// TwinCAT 3 PLC project Motion
// ProgramVersion: 3.1.4022.7
// libraries:
//   LCLS General, * (SLAC)
//   lcls-twincat-motion, * (SLAC)
//   PMPS, * (SLAC - LCLS)
//   Tc2_MC2, * (Beckhoff Automation GmbH)
//   Tc2_Standard, * (Beckhoff Automation GmbH)
//   Tc2_System, * (Beckhoff Automation GmbH)
//   Tc3_Module, * (Beckhoff Automation GmbH)
//   TcUnit, * (www.tcunit.org)
// project tree:
//   DUTs/ DUT_SensorHGS.TcDUT, DUT_Sensor.TcDUT (not stored)
//   GVLs/ GVL_Main.TcGVL, GVL_PMPS.TcGVL, GVL_Sensor.TcGVL (not stored)
//   / PlcTask.TcTTO
//   POUs/ FB_2AxesTrans.TcPOU, FB_3AxesJack.TcPOU, PRG1_MAIN_PlcTask.TcPOU, FB_Slits.TcPOU, PRG_2Theta.TcPOU, PRG_DET_ARM.TcPOU, PRG_DET_CHAMBER.TcPOU, PRG_DET_SLIT.TcPOU, PRG_DET_FRAME.TcPOU, PRG_OPT.TcPOU, PRG_OPT_XPM.TcPOU, PRG_OPT_SLITS.TcPOU, PRG_OPT_YG.TcPOU, PRG_Sensor.TcPOU
// real-time tasks:
//   TASK PlcTask: cycle T#10ms, priority 20, ADS port 350
// motion (NC):
//   TASK NC-Task 1 SAF: cycle T#2ms, priority 4, ADS port 501
//   TASK NC-Task 1 SVB: cycle T#10ms, priority 8, ADS port 511
//   AXIS ServoDrive (id 1)
//     General: UnitName=deg
//     Dynamic: AccelerationMaximum=10, DecelerationMaximum=10, Acceleration=0.5, Deceleration=0.5, Jerk=1
//     Velo: RefSearch=0.25, RefSync=0.25, SlowManual=0.25, FastManual=0.25, Maximum=0.25
//     OtherSettings: AllowMotionCmdToSlave=true, PulseDistancePos=1, PulseDistanceNeg=1
//     encoder EncType=19
//       EncPara: ScaleFactorNumerator=3.001664895e-06, Offset=-76.2211171, MaxCount=#xffffffff
//         SoftEndMinControl: Enable=true, Range=42
//         SoftEndMaxControl: Enable=true, Range=149.4
//     drive DrvType=16
//       DrvPara: MaxCount=#xffffffff, DriveControlDWord=#x00020100
//         Analog: VeloReferenz=0.25, ScaleFactorActTorque=0.1
//         TimeComp: TaskDelayCycles=1
//     controller CtrType=2
//       CtrPara: PriorControlFactor=1
//         PosDiffControl: Range=2
//         PID: DeadBandPosition=0.05
//         Observer: BandWidth=20
//   AXIS Stepper (id 27)
//     General: UnitName=deg
//     Dynamic: AccelerationMaximum=1.5, DecelerationMaximum=1.5, Acceleration=1.4, Deceleration=0.7, Jerk=2.8
//     Velo: Maximum=0.7
//     PositionAreaControl: Range=0.5
//     TargetPosControl: Range=0.1
//     OtherSettings: AllowMotionCmdToSlave=true
//     encoder EncType=29
//       EncPara: ScaleFactorNumerator=3.001664895e-06, Offset=13.6052237, MaxCount=#xffffffff
//         SoftEndMinControl: Enable=true, Range=42
//         SoftEndMaxControl: Enable=true, Range=149.4
//         Inc: RefSoftSyncMask=#x0000ffff
//     drive DrvType=24
//       Analog: VeloReferenz=0.715862885, ScaleFactorActTorque=0.1
//       TimeComp: TaskDelayCycles=1
//     controller CtrType=2
//       CtrPara: PriorControlFactor=1
//         PosDiffControl: Range=0.5
//         PID: DeadBandPosition=0.05
//         Observer: BandWidth=20
//   AXIS XS1 (id 11)
//     Dynamic: AccelerationMaximum=20, DecelerationMaximum=20, Acceleration=10, Deceleration=10, Jerk=100
//     Velo: Maximum=1
//     PositionAreaControl: Range=1
//     TargetPosControl: Range=0.05
//     OtherSettings: AllowMotionCmdToSlave=true
//     encoder EncType=29
//       EncPara: ScaleFactorNumerator=5e-05, Offset=-48.701, MaxCount=#xffffffff
//         SoftEndMinControl: Enable=true, Range=-25
//         SoftEndMaxControl: Enable=true, Range=25
//         Inc: RefSoftSyncMask=#x0000ffff
//     drive DrvType=24
//       Analog: VeloReferenz=1, ScaleFactorActTorque=0.1
//       TimeComp: TaskDelayCycles=1
//     controller CtrType=2
//       CtrPara: PriorControlFactor=1
//         PosDiffControl: Range=1
//         PID: DeadBandPosition=0.0002
//         Observer: BandWidth=20
//   AXIS XS2 (id 12)
//     Dynamic: AccelerationMaximum=20, DecelerationMaximum=20, Acceleration=10, Deceleration=10, Jerk=100
//     Velo: Maximum=1
//     PositionAreaControl: Range=1
//     TargetPosControl: Range=0.05
//     OtherSettings: AllowMotionCmdToSlave=true
//     encoder EncType=29
//       EncPara: ScaleFactorNumerator=5e-05, Offset=-50.138, MaxCount=#xffffffff
//         SoftEndMinControl: Enable=true, Range=-25
//         SoftEndMaxControl: Enable=true, Range=25
//         Inc: RefSoftSyncMask=#x0000ffff
//     drive DrvType=24
//       Analog: VeloReferenz=1, ScaleFactorActTorque=0.1
//       TimeComp: TaskDelayCycles=1
//     controller CtrType=2
//       CtrPara: PriorControlFactor=1
//         PosDiffControl: Range=1
//         PID: DeadBandPosition=0.0002
//         Observer: BandWidth=20
//   AXIS YS1 (id 13)
//     Dynamic: AccelerationMaximum=20, DecelerationMaximum=20, Acceleration=10, Deceleration=10, Jerk=100
//     Velo: Maximum=1
//     PositionAreaControl: Range=1
//     TargetPosControl: Range=0.05
//     OtherSettings: AllowMotionCmdToSlave=true
//     encoder EncType=29
//       EncPara: ScaleFactorNumerator=5e-05, Offset=-53.276, MaxCount=#xffffffff
//         SoftEndMinControl: Enable=true, Range=-25
//         SoftEndMaxControl: Enable=true, Range=25
//         Inc: RefSoftSyncMask=#x0000ffff
//     drive DrvType=24
//       Analog: VeloReferenz=1, ScaleFactorActTorque=0.1
//       TimeComp: TaskDelayCycles=1
//     controller CtrType=2
//       CtrPara: PriorControlFactor=1
//         PosDiffControl: Range=1
//         PID: DeadBandPosition=0.0002
//         Observer: BandWidth=20
//   AXIS YS2 (id 14)
//     Dynamic: AccelerationMaximum=20, DecelerationMaximum=20, Acceleration=10, Deceleration=10, Jerk=100
//     Velo: Maximum=1
//     PositionAreaControl: Range=1
//     TargetPosControl: Range=0.05
//     OtherSettings: AllowMotionCmdToSlave=true
//     encoder EncType=29
//       EncPara: ScaleFactorNumerator=5e-05, Offset=-50.673, MaxCount=#xffffffff
//         SoftEndMinControl: Enable=true, Range=-25
//         SoftEndMaxControl: Enable=true, Range=25
//         Inc: RefSoftSyncMask=#x0000ffff
//     drive DrvType=24
//       Analog: VeloReferenz=1, ScaleFactorActTorque=0.1
//       TimeComp: TaskDelayCycles=1
//     controller CtrType=2
//       CtrPara: PriorControlFactor=1
//         PosDiffControl: Range=1
//         PID: DeadBandPosition=0.0002
//         Observer: BandWidth=20
//   AXIS YG1 (id 17)
//     Dynamic: AccelerationMaximum=0.4, DecelerationMaximum=0.4, Acceleration=0.2, Deceleration=0.2, Jerk=0.4
//     Velo: SlowManual=0.25, FastManual=0.5, Maximum=0.05
//     PositionAreaControl: Range=0.1
//     TargetPosControl: Range=0.05
//     BacklashCompensation: Range=0.025
//     OtherSettings: AllowMotionCmdToSlave=true, PulseDistancePos=1, PulseDistanceNeg=1
//     encoder EncType=29
//       EncPara: ScaleFactorNumerator=5e-06, Offset=-48.289375, MaxCount=#xffffffff
//         SoftEndMinControl: Enable=true, Range=-7.2
//         SoftEndMaxControl: Enable=true, Range=7.2
//         Inc: RefSoftSyncMask=#x0000ffff
//     drive DrvType=24
//       Analog: VeloReferenz=0.1, ScaleFactorActTorque=0.1
//       TimeComp: TaskDelayCycles=1
//     controller CtrType=2
//       CtrPara: PriorControlFactor=1
//         PosDiffControl: Range=2
//         PID: DeadBandPosition=0.0001
//         Observer: BandWidth=20
//   AXIS YG2 (id 18)
//     Dynamic: AccelerationMaximum=0.4, DecelerationMaximum=0.4, Acceleration=0.2, Deceleration=0.2, Jerk=0.4
//     Velo: Maximum=0.05
//     PositionAreaControl: Range=0.5
//     TargetPosControl: Range=0.05
//     OtherSettings: AllowMotionCmdToSlave=true
//     encoder EncType=29
//       EncPara: ScaleFactorNumerator=5e-06, Offset=-49.0846, MaxCount=#xffffffff
//         SoftEndMinControl: Enable=true, Range=-7.2
//         SoftEndMaxControl: Enable=true, Range=-7.2
//         Inc: RefSoftSyncMask=#x0000ffff
//     drive DrvType=24
//       Analog: VeloReferenz=0.1, ScaleFactorActTorque=0.1
//       TimeComp: TaskDelayCycles=1
//     controller CtrType=2
//       CtrPara: PriorControlFactor=1
//         PosDiffControl: Range=2
//         PID: DeadBandPosition=0.0001
//         Observer: BandWidth=20
//   AXIS YG3 (id 19)
//     Dynamic: AccelerationMaximum=0.4, DecelerationMaximum=0.4, Acceleration=0.2, Deceleration=0.2, Jerk=0.4
//     Velo: Maximum=0.05
//     PositionAreaControl: Range=0.1
//     TargetPosControl: Range=0.05
//     OtherSettings: AllowMotionCmdToSlave=true
//     encoder EncType=29
//       EncPara: ScaleFactorNumerator=5e-06, Offset=-49.5733, MaxCount=#xffffffff
//         SoftEndMinControl: Enable=true, Range=-7.2
//         SoftEndMaxControl: Enable=true, Range=7.2
//         Inc: RefSoftSyncMask=#x0000ffff
//     drive DrvType=24
//       Analog: VeloReferenz=0.1, ScaleFactorActTorque=0.1
//       TimeComp: TaskDelayCycles=1
//     controller CtrType=2
//       CtrPara: PriorControlFactor=1
//         PosDiffControl: Range=2
//         PID: DeadBandPosition=0.0001
//         Observer: BandWidth=20
//   AXIS RxG (id 15)
//     General: UnitName=mrad
//     Dynamic: AccelerationMaximum=2, DecelerationMaximum=2, Acceleration=2, Deceleration=2, Jerk=10
//     Velo: Maximum=1.29
//     TargetPosControl: Range=0.01
//     OtherSettings: AllowMotionCmdToSlave=true
//     encoder EncType=19
//       EncPara: ScaleFactorNumerator=1.462918079, ScaleFactorDenominator=1000000, Offset=2351.695, MaxCount=#xffffffff
//         SoftEndMinControl: Enable=true, Range=-17.5
//         SoftEndMaxControl: Enable=true, Range=87.5
//         Inc: RefSoftSyncMask=#x0000ffff
//     drive DrvType=24
//       Analog: VeloReferenz=1.29032258064516, ScaleFactorActTorque=0.1
//       TimeComp: TaskDelayCycles=1
//     controller CtrType=2
//       CtrPara: PriorControlFactor=1
//         PosDiffControl: Range=0.5
//         PID: DeadBandPosition=5e-05
//         Observer: BandWidth=20
//   AXIS XG (id 16)
//     Dynamic: AccelerationMaximum=40, DecelerationMaximum=40, Acceleration=20, Deceleration=20, Jerk=20000
//     Velo: Maximum=2
//     TargetPosControl: Range=0.1
//     OtherSettings: AllowMotionCmdToSlave=true
//     encoder EncType=29
//       EncPara: ScaleFactorNumerator=5e-05, Offset=-123.91085, MaxCount=#xffffffff
//         SoftEndMinControl: Enable=true, Range=-95
//         SoftEndMaxControl: Enable=true, Range=95
//         Inc: RefSoftSyncMask=#x0000ffff
//     drive DrvType=24
//       Analog: VeloReferenz=10, ScaleFactorActTorque=0.1
//       TimeComp: TaskDelayCycles=1
//     controller CtrType=2
//       CtrPara: PriorControlFactor=1
//         PID: DeadBandPosition=0.001
//         Observer: BandWidth=20
//   AXIS XPM1 (id 20)
//     Dynamic: AccelerationMaximum=20, DecelerationMaximum=20, Acceleration=20, Deceleration=20, Jerk=400
//     Velo: RefSearch=1, RefSync=1, SlowManual=0.5, FastManual=1, Maximum=0.1
//     PositionAreaControl: Range=1
//     TargetPosControl: Range=0.02
//     OtherSettings: AllowMotionCmdToSlave=true, PulseDistancePos=1, PulseDistanceNeg=1
//     encoder EncType=29
//       EncPara: ScaleFactorNumerator=5e-05, Offset=-50.788, MaxCount=#xffffffff
//         SoftEndMinControl: Enable=true, Range=-17.5
//         SoftEndMaxControl: Enable=true, Range=17.5
//         Inc: RefSoftSyncMask=#x0000ffff
//     drive DrvType=24
//       Analog: VeloReferenz=0.2, ScaleFactorActTorque=0.1
//       TimeComp: TaskDelayCycles=1
//     controller CtrType=2
//       CtrPara: PriorControlFactor=1
//         PosDiffControl: Range=0.5, Time=0.01
//         PID: DeadBandPosition=0.0001
//         Observer: BandWidth=20
//   AXIS XPM2 (id 21)
//     Dynamic: AccelerationMaximum=20, DecelerationMaximum=20, Acceleration=20, Deceleration=20, Jerk=400
//     Velo: RefSearch=1, RefSync=1, SlowManual=0.5, FastManual=1, Maximum=0.1
//     PositionAreaControl: Range=1
//     TargetPosControl: Range=0.02
//     OtherSettings: AllowMotionCmdToSlave=true, PulseDistancePos=1, PulseDistanceNeg=1
//     encoder EncType=29
//       EncPara: ScaleFactorNumerator=5e-05, Offset=-48.577, MaxCount=#xffffffff
//         SoftEndMinControl: Enable=true, Range=-17.5
//         SoftEndMaxControl: Enable=true, Range=17.5
//         Inc: RefSoftSyncMask=#x0000ffff
//     drive DrvType=24
//       Analog: VeloReferenz=0.2, ScaleFactorActTorque=0.1
//       TimeComp: TaskDelayCycles=1
//     controller CtrType=2
//       CtrPara: PriorControlFactor=1
//         PosDiffControl: Range=1
//         PID: DeadBandPosition=0.0001
//         Observer: BandWidth=20
//   AXIS RzPM (id 22)
//     General: UnitName=mrad
//     Dynamic: AccelerationMaximum=2.6, DecelerationMaximum=2.6, Acceleration=2.6, Deceleration=2.6, Jerk=52
//     Velo: RefSearch=2000, RefSync=2000, SlowManual=1000, FastManual=2000, Maximum=0.2
//     PositionAreaControl: Range=0.1
//     TargetPosControl: Range=0.01
//     OtherSettings: AllowMotionCmdToSlave=true
//     encoder EncType=29
//       EncPara: ScaleFactorNumerator=0.299580587, ScaleFactorDenominator=1000, Offset=-205.8664, MaxCount=#xffffffff
//         SoftEndMinControl: Enable=true, Range=-60
//         SoftEndMaxControl: Enable=true, Range=60
//         Inc: RefSoftSyncMask=#x0000ffff
//     drive DrvType=24
//       Analog: VeloReferenz=1.3333333, ScaleFactorActTorque=0.1
//       TimeComp: TaskDelayCycles=1
//     controller CtrType=2
//       CtrPara: PriorControlFactor=1
//         PosDiffControl: Range=0.1
//         PID: DeadBandPosition=0.0005
//         Observer: BandWidth=20
//   AXIS YDF1 (id 23)
//     Dynamic: AccelerationMaximum=1, DecelerationMaximum=1, Acceleration=0.8, Deceleration=0.8, Jerk=3.2
//     Velo: FastManual=0, Maximum=0.05
//     PositionAreaControl: Range=0.5
//     OtherSettings: AllowMotionCmdToSlave=true
//     encoder EncType=1
//       EncPara: ScaleFactorNumerator=1
//         SoftEndMinControl: Enable=true, Range=-0.5
//         SoftEndMaxControl: Range=21.5
//         Inc: RefSoftSyncMask=#x0000ffff
//     drive DrvType=24
//       Analog: VeloReferenz=0.333336, ScaleFactorActTorque=0.1
//       TimeComp: TaskDelayCycles=1
//     controller CtrType=1
//       CtrPara: PriorControlFactor=1
//         PosDiffControl: Range=0.5
//         Observer: BandWidth=20
//   AXIS YDF2 (id 24)
//     Dynamic: AccelerationMaximum=1, DecelerationMaximum=1, Acceleration=0.8, Deceleration=0.8, Jerk=3.2
//     Velo: FastManual=0, Maximum=0.05
//     PositionAreaControl: Range=0.5
//     OtherSettings: AllowMotionCmdToSlave=true
//     encoder EncType=1
//       EncPara: ScaleFactorNumerator=4.2e-05
//         SoftEndMinControl: Enable=true, Range=-0.5
//         SoftEndMaxControl: Range=21.5
//         Inc: RefSoftSyncMask=#x0000ffff
//     drive DrvType=24
//       Analog: VeloReferenz=0.333336, ScaleFactorActTorque=0.1
//       TimeComp: TaskDelayCycles=1
//     controller CtrType=1
//       CtrPara: PriorControlFactor=1
//         PosDiffControl: Range=0.5
//         Observer: BandWidth=20
//   AXIS YDF3 (id 25)
//     Dynamic: AccelerationMaximum=1, DecelerationMaximum=1, Acceleration=0.8, Deceleration=0.8, Jerk=3.2
//     Velo: FastManual=0, Maximum=0.05
//     PositionAreaControl: Range=0.5
//     OtherSettings: AllowMotionCmdToSlave=true
//     encoder EncType=1
//       EncPara: ScaleFactorNumerator=4.2e-05
//         SoftEndMinControl: Enable=true, Range=-0.5
//         SoftEndMaxControl: Enable=true, Range=21.5
//         Inc: RefSoftSyncMask=#x0000ffff
//     drive DrvType=24
//       Analog: VeloReferenz=0.333336, ScaleFactorActTorque=0.1
//       TimeComp: TaskDelayCycles=1
//     controller CtrType=1
//       CtrPara: PriorControlFactor=1
//         PosDiffControl: Range=0.5
//         Observer: BandWidth=20
//   AXIS XSDC1 (id 2)
//     Dynamic: AccelerationMaximum=20, DecelerationMaximum=20, Acceleration=10, Deceleration=10, Jerk=100
//     Velo: Maximum=1
//     PositionAreaControl: Range=1
//     TargetPosControl: Range=0.1
//     OtherSettings: AllowMotionCmdToSlave=true
//     encoder EncType=29
//       EncPara: ScaleFactorNumerator=5e-05, Offset=-49.035, MaxCount=#xffffffff
//         SoftEndMinControl: Enable=true, Range=-25
//         SoftEndMaxControl: Enable=true, Range=25
//         Inc: RefSoftSyncMask=#x0000ffff
//     drive DrvType=24
//       Analog: VeloReferenz=1, ScaleFactorActTorque=0.1
//       TimeComp: TaskDelayCycles=1
//     controller CtrType=2
//       CtrPara: PriorControlFactor=1
//         PosDiffControl: Range=1
//         PID: DeadBandPosition=0.0002
//         Observer: BandWidth=20
//   AXIS XSDC2 (id 3)
//     Dynamic: AccelerationMaximum=20, DecelerationMaximum=20, Acceleration=10, Deceleration=10, Jerk=100
//     Velo: Maximum=1
//     PositionAreaControl: Range=1
//     TargetPosControl: Range=0.1
//     OtherSettings: AllowMotionCmdToSlave=true
//     encoder EncType=29
//       EncPara: ScaleFactorNumerator=5e-05, Offset=-49.27, MaxCount=#xffffffff
//         SoftEndMinControl: Enable=true, Range=-25
//         SoftEndMaxControl: Enable=true, Range=25
//         Inc: RefSoftSyncMask=#x0000ffff
//     drive DrvType=24
//       Analog: VeloReferenz=1, ScaleFactorActTorque=0.1
//       TimeComp: TaskDelayCycles=1
//     controller CtrType=2
//       CtrPara: PriorControlFactor=1
//         PosDiffControl: Range=1
//         PID: DeadBandPosition=0.0002
//         Observer: BandWidth=20
//   AXIS YSDC1 (id 4)
//     Dynamic: AccelerationMaximum=20, DecelerationMaximum=20, Acceleration=10, Deceleration=10, Jerk=100
//     Velo: Maximum=1
//     PositionAreaControl: Range=1
//     TargetPosControl: Range=0.1
//     OtherSettings: AllowMotionCmdToSlave=true
//     encoder EncType=29
//       EncPara: ScaleFactorNumerator=5e-05, Offset=-51.43, MaxCount=#xffffffff
//         SoftEndMinControl: Enable=true, Range=-25
//         SoftEndMaxControl: Enable=true, Range=25
//         Inc: RefSoftSyncMask=#x0000ffff
//     drive DrvType=24
//       Analog: VeloReferenz=1, ScaleFactorActTorque=0.1
//       TimeComp: TaskDelayCycles=1
//     controller CtrType=2
//       CtrPara: PriorControlFactor=1
//         PosDiffControl: Range=1
//         PID: DeadBandPosition=0.0002
//         Observer: BandWidth=20
//   AXIS YSDC2 (id 5)
//     Dynamic: AccelerationMaximum=20, DecelerationMaximum=20, Acceleration=10, Deceleration=10, Jerk=100
//     Velo: Maximum=1
//     PositionAreaControl: Range=1
//     TargetPosControl: Range=0.1
//     OtherSettings: AllowMotionCmdToSlave=true
//     encoder EncType=29
//       EncPara: ScaleFactorNumerator=5e-05, Offset=-49.4945, MaxCount=#xffffffff
//         SoftEndMinControl: Enable=true, Range=-25
//         SoftEndMaxControl: Enable=true, Range=25
//         Inc: RefSoftSyncMask=#x0000ffff
//     drive DrvType=24
//       Analog: VeloReferenz=1, ScaleFactorActTorque=0.1
//       TimeComp: TaskDelayCycles=1
//     controller CtrType=2
//       CtrPara: PriorControlFactor=1
//         PosDiffControl: Range=1
//         PID: DeadBandPosition=0.0002
//         Observer: BandWidth=20
//   AXIS XDC (id 6)
//     Dynamic: AccelerationMaximum=0.5, DecelerationMaximum=0.5, Acceleration=0.5, Deceleration=0.5, Jerk=0.5
//     Velo: RefSearch=0.5, RefSync=0.5, SlowManual=0.5, FastManual=1, Maximum=1
//     PositionAreaControl: Range=1
//     TargetPosControl: Range=0.5
//     OtherSettings: AllowMotionCmdToSlave=true, PulseDistancePos=1, PulseDistanceNeg=1
//     encoder EncType=29
//       EncPara: ScaleFactorNumerator=5e-05, Offset=-29.66, MaxCount=#xffffffff
//         SoftEndMinControl: Enable=true, Range=-12
//         SoftEndMaxControl: Enable=true, Range=12
//         Inc: RefSoftSyncMask=#x0000ffff
//     drive DrvType=24
//       Analog: VeloReferenz=10, ScaleFactorActTorque=0.1
//       TimeComp: TaskDelayCycles=1
//     controller CtrType=1
//       CtrPara: PriorControlFactor=1
//         PosDiffControl: Range=1
//         Observer: BandWidth=20
//   AXIS RyDC (id 7)
//     General: UnitName=mrad
//     Dynamic: AccelerationMaximum=4, DecelerationMaximum=4, Acceleration=4, Deceleration=4, Jerk=6
//     Velo: RefSearch=200, RefSync=200, SlowManual=500, FastManual=1000, Maximum=1
//     PositionAreaControl: Range=2
//     TargetPosControl: Range=0.02
//     OtherSettings: AllowMotionCmdToSlave=true, PulseDistancePos=100, PulseDistanceNeg=100
//     encoder EncType=29
//       EncPara: ScaleFactorNumerator=5e-05, ScaleFactorDenominator=0.2454, Offset=-138.3455583, MaxCount=#xffffffff
//         SoftEndMinControl: Enable=true, Range=-85
//         SoftEndMaxControl: Enable=true, Range=85
//         Inc: RefSoftSyncMask=#x0000ffff
//     drive DrvType=24
//       Analog: VeloReferenz=40.74979625, ScaleFactorActTorque=0.1
//       TimeComp: TaskDelayCycles=1
//     controller CtrType=1
//       CtrPara: PriorControlFactor=1
//         PosDiffControl: Range=2
//         Observer: BandWidth=20
//   AXIS ZDC (id 8)
//     Dynamic: AccelerationMaximum=2, DecelerationMaximum=2, Acceleration=2, Deceleration=2, Jerk=4
//     Velo: RefSearch=0.5, RefSync=0.5, SlowManual=0.5, FastManual=1, Maximum=0.25
//     PositionAreaControl: Range=1
//     TargetPosControl: Range=1
//     OtherSettings: AllowMotionCmdToSlave=true, PulseDistancePos=1, PulseDistanceNeg=1
//     encoder EncType=29
//       EncPara: ScaleFactorNumerator=5e-05, Offset=-29.48, MaxCount=#xffffffff
//         SoftEndMinControl: Enable=true, Range=-5.05
//         SoftEndMaxControl: Enable=true, Range=5.05
//         Inc: RefSoftSyncMask=#x0000ffff
//     drive DrvType=24
//       Analog: VeloReferenz=20, ScaleFactorActTorque=0.1
//       TimeComp: TaskDelayCycles=1
//     controller CtrType=1
//       CtrPara: PriorControlFactor=1
//         PosDiffControl: Range=1
//         Observer: BandWidth=20
//   AXIS YF1 (id 9)
//     Dynamic: AccelerationMaximum=8, DecelerationMaximum=8, Acceleration=5, Deceleration=5, Jerk=12.5
//     Velo: RefSearch=0.5, RefSync=0.5, SlowManual=0.5, FastManual=1, Maximum=2
//     PositionAreaControl: Range=2
//     TargetPosControl: Range=1
//     OtherSettings: AllowMotionCmdToSlave=true
//     encoder EncType=29
//       EncPara: ScaleFactorNumerator=5e-05, Offset=-993.1032, MaxCount=#xffffffff
//         SoftEndMinControl: Enable=true, Range=-925
//         SoftEndMaxControl: Enable=true, Range=-225
//         Inc: RefSoftSyncMask=#x0000ffff
//     drive DrvType=24
//       Analog: VeloReferenz=2, ScaleFactorActTorque=0.1
//       TimeComp: TaskDelayCycles=1
//     controller CtrType=1
//       CtrPara: PriorControlFactor=1
//         PosDiffControl: Range=2
//         Observer: BandWidth=20
//   AXIS YF2 (id 10)
//     Dynamic: AccelerationMaximum=8, DecelerationMaximum=8, Acceleration=4, Deceleration=4, Jerk=8
//     Velo: RefSearch=0.5, RefSync=0.5, SlowManual=0.5, FastManual=1, Maximum=2
//     PositionAreaControl: Range=2
//     TargetPosControl: Range=1
//     OtherSettings: AllowMotionCmdToSlave=true
//     encoder EncType=29
//       EncPara: ScaleFactorNumerator=5e-05, Offset=-993.2193, MaxCount=#xffffffff
//         SoftEndMinControl: Enable=true, Range=-925
//         SoftEndMaxControl: Enable=true, Range=-225
//         Inc: RefSoftSyncMask=#x0000ffff
//     drive DrvType=24
//       Analog: VeloReferenz=2, ScaleFactorActTorque=0.1
//       TimeComp: TaskDelayCycles=1
//     controller CtrType=1
//       CtrPara: PriorControlFactor=1
//         PosDiffControl: Range=2
//         Observer: BandWidth=20
//   AXIS ZF (id 26)
//     Dynamic: AccelerationMaximum=4, DecelerationMaximum=4, Acceleration=4, Deceleration=4, Jerk=8
//     Velo: RefSearch=0.5, RefSync=0.5, SlowManual=0.5, FastManual=1, Maximum=2
//     PositionAreaControl: Range=2
//     TargetPosControl: Range=0.5
//     BacklashCompensation: Enable=true, Range=0.003
//     OtherSettings: AllowMotionCmdToSlave=true
//     encoder EncType=29
//       EncPara: ScaleFactorNumerator=5e-05, Offset=2579.4011, MaxCount=#xffffffff
//         SoftEndMinControl: Enable=true, Range=2650
//         SoftEndMaxControl: Enable=true, Range=3600
//         Inc: RefSoftSyncMask=#x0000ffff
//     drive DrvType=24
//       Analog: VeloReferenz=4, ScaleFactorActTorque=0.1
//       TimeComp: TaskDelayCycles=1
//     controller CtrType=2
//       CtrPara: PriorControlFactor=1
//         PosDiffControl: Range=2
//         PID: AccKa=0.1, DeadBandPosition=0.005
//         Observer: BandWidth=20
// I/O:
//   DEVICE CX2020 (EtherCAT), AmsNetId 5.88.101.160.2.1
//     Term 1 (EK1200) [EK1200-5000 EtherCAT Power supply (2A E-Bus)]
//       Term 2 (EK1122) [EK1122 2 port EtherCAT junction]
//         Rack#1C_ServoDR (NCR-HD Series) [NCR-HD Series AC Servo Drive] (disabled)
//         Rack#1A-01 Coupler (EK1100) [EK1100 EtherCAT Coupler (2A E-Bus)]
//           Rack#1A-02 SFIN (EL1918) [EL1918, 8Ch. Safety Input 24V, TwinSAFE]
//             modules: Module 2 (FSLOGIC)
//           Rack#1A-03 SFOUT(EL2912) [EL2912, 2Ch. Safety Output 24V, 2A, TwinSAFE]
//             modules: Module 1 (FSOE), Module 2 (FSOUT), Module 3 (DEVICEIO), Module 4 (FSLOGIC)
//           Rack#1A-04 DR_2Th (EL7047) [EL7047 1Ch. Stepper motor output stage (50V, 5A)]
//           Rack#1A-05 MB_2Th (EL2602) [EL2602 2Ch. Relay Output, NO (230V AC / 30V DC)]
//           Rack#1A-06 ENC_2Th (EL5042) [EL5042 2Ch. BiSS-C Encoder]
//           Rack#1A-07 ECAT Extension (EK1110) [EK1110 EtherCAT extension]
//         BOX-01 Coupler (EK1100) [EK1100 EtherCAT Coupler (2A E-Bus)]
//           BOX-02 SFIN(EL1904) [EL1904, 4 Ch. Safety Input 24V, TwinSAFE]
//             modules: Module 1 (FSOES)
//           BOX-03 ENC_X1_X2 (EL5042) [EL5042 2Ch. BiSS-C Encoder]
//           BOX-04 ENC_Y1_Y2 (EL5042) [EL5042 2Ch. BiSS-C Encoder]
//           BOX-05 ENC_XDC_RyDC (EL5042) [EL5042 2Ch. BiSS-C Encoder]
//           BOX-06 ENC_ZDC_YF1 (EL5042) [EL5042 2Ch. BiSS-C Encoder]
//           BOX-07 ENC_YF2_ZF (EL5042) [EL5042 2Ch. BiSS-C Encoder]
//           BOX-08 CP_SDC (EL9221-5000) [EL9221-5000 Overcurrent protection 24V DC, 1Ch., max. 10A, adjustable]
//           BOX-09 DR_XSDC1 (EL7041-0052) [EL7041-0052 1Ch. Stepper motor output stage (50V, 5A)]
//           BOX-10 DR_XSDC2 (EL7041-0052) [EL7041-0052 1Ch. Stepper motor output stage (50V, 5A)]
//           BOX-11 DR_YSDC1 (EL7041-0052) [EL7041-0052 1Ch. Stepper motor output stage (50V, 5A)]
//           BOX-12 DR_YSDC2 (EL7041-0052) [EL7041-0052 1Ch. Stepper motor output stage (50V, 5A)]
//           BOX-13 CP_DC (EL9221-5000) [EL9221-5000 Overcurrent protection 24V DC, 1Ch., max. 10A, adjustable]
//           BOX-14 DR_XDC (EL7041-0052) [EL7041-0052 1Ch. Stepper motor output stage (50V, 5A)]
//           BOX-15 DR_RyDC (EL7041-0052) [EL7041-0052 1Ch. Stepper motor output stage (50V, 5A)]
//           BOX-16 DR_ZDC (EL7041-0052) [EL7041-0052 1Ch. Stepper motor output stage (50V, 5A)]
//           BOX-17 Ebus Reflesh (EL9410) [EL9410 E-Bus Power Supplier  (Diagnostics)]
//           BOX-18 CP_YF1_YF2 (EL9221-5000) [EL9221-5000 Overcurrent protection 24V DC, 1Ch., max. 10A, adjustable]
//           BOX-19 MB_YF1_YF2 (EL2602) [EL2602 2Ch. Relay Output, NO (230V AC / 30V DC)]
//           BOX-20 DR_YF1 (EL7047) [EL7047 1Ch. Stepper motor output stage (50V, 5A)]
//           BOX-21 DR_YF2 (EL7047) [EL7047 1Ch. Stepper motor output stage (50V, 5A)]
//           BOX-22 EtherCAT Extension (EK1110) [EK1110 EtherCAT extension]
//         Rack#2A-01 Coupler (EK1100) [EK1100 EtherCAT Coupler (2A E-Bus)]
//           Rack#2A-02 CP_SLIT (EL9221-5000) [EL9221-5000 Overcurrent protection 24V DC, 1Ch., max. 10A, adjustable]
//           Rack#2A-03 DR_XS1 (EL7041-0052) [EL7041-0052 1Ch. Stepper motor output stage (50V, 5A)]
//           Rack#2A-04 DR_XS2 (EL7041-0052) [EL7041-0052 1Ch. Stepper motor output stage (50V, 5A)]
//           Rack#2A-05 DR_YS1 (EL7041-0052) [EL7041-0052 1Ch. Stepper motor output stage (50V, 5A)]
//           Rack#2A-06 DR_YS2 (EL7041-0052) [EL7041-0052 1Ch. Stepper motor output stage (50V, 5A)]
//           Rack#2A-07 CP_G (EL9221-5000) [EL9221-5000 Overcurrent protection 24V DC, 1Ch., max. 10A, adjustable]
//           Rack#2A-08 DR_RxG (EL7041-0052) [EL7041-0052 1Ch. Stepper motor output stage (50V, 5A)]
//           Rack#2A-09 DR_XG (EL7041-0052) [EL7041-0052 1Ch. Stepper motor output stage (50V, 5A)]
//           Rack#2A-10 DR_YG1 (EL7041-0052) [EL7041-0052 1Ch. Stepper motor output stage (50V, 5A)]
//           Rack#2A-11 DR_YG2 (EL7041-0052) [EL7041-0052 1Ch. Stepper motor output stage (50V, 5A)]
//           Rack#2A-12 DR_YG3 (EL7041-0052) [EL7041-0052 1Ch. Stepper motor output stage (50V, 5A)]
//           Rack#2A-13 CP_PM (EL9221-5000) [EL9221-5000 Overcurrent protection 24V DC, 1Ch., max. 10A, adjustable]
//           Rack#2A-14 DR_XPM1 (EL7041-0052) [EL7041-0052 1Ch. Stepper motor output stage (50V, 5A)]
//           Rack#2A-15 DR_XPM2 (EL7041-0052) [EL7041-0052 1Ch. Stepper motor output stage (50V, 5A)]
//           Rack#2A-16 DR_RzPM (EL7041-0052) [EL7041-0052 1Ch. Stepper motor output stage (50V, 5A)]
//           Rack#2A-17 EtherCAT Extension (EK1110) [EK1110 EtherCAT extension]
//         Rack#2B-01 Coupler (EK1100) [EK1100 EtherCAT Coupler (2A E-Bus)]
//           Rack#2B-02 KTC (EL3314) [EL3314 4Ch. Ana. Input Thermocouple (TC)]
//           Rack#2B-03 AI_TiltSensor (EL3174-0002) [EL3174-0002 4Ch. Ana. Input +/-10V, +/-20mA 16 Bit, Isolated Channels]
//           Rack#2B-04 PS_P (EL3064) [EL3064 4Ch. Ana. Input 0-10V]
//           Rack#2B-05 SV_AIR (EL2004) [EL2004 4Ch. Dig. Output 24V, 0.5A]
//           Rack#2B-06 SFIN (EL1918) [EL1918, 8Ch. Safety Input 24V, TwinSAFE]
//             modules: Module 1 (FSOE), Module 2 (FSLOGIC)
//           Rack#2B-07 ENC_X1_X2 (EL5042) [EL5042 2Ch. BiSS-C Encoder]
//           Rack#2B-08 ENC_Y1_Y2 (EL5042) [EL5042 2Ch. BiSS-C Encoder]
//           Rack#2B-09 ENC_RxG_XG (EL5042) [EL5042 2Ch. BiSS-C Encoder]
//           Rack#2B-10 ENC_YG1_YG2 (EL5042) [EL5042 2Ch. BiSS-C Encoder]
//           Rack#2B-11 ENC_YG3_X1PM (EL5042) [EL5042 2Ch. BiSS-C Encoder]
//           Rack#2B-12 ENC_X2PM_RzPM (EL5042) [EL5042 2Ch. BiSS-C Encoder]
//           Rack#2B-13 PWS_EBUS (EL9410) [EL9410 E-Bus Power Supplier  (Diagnostics)]
//           Rack#2B-14 CP_YDF (EL9221-5000) [EL9221-5000 Overcurrent protection 24V DC, 1Ch., max. 10A, adjustable]
//           Rack#2B-15 DR_YDF1 (EL7041-0052) [EL7041-0052 1Ch. Stepper motor output stage (50V, 5A)]
//           Rack#2B-16 DR_YDF2 (EL7041-0052) [EL7041-0052 1Ch. Stepper motor output stage (50V, 5A)]
//           Rack#2B-17 CP_YDF_ZF (EL9221-5000) [EL9221-5000 Overcurrent protection 24V DC, 1Ch., max. 10A, adjustable]
//           Rack#2B-18 MB_ZF (EL2602) [EL2602 2Ch. Relay Output, NO (230V AC / 30V DC)]
//           Rack#2B-19 DR_YDF3 (EL7041-0052) [EL7041-0052 1Ch. Stepper motor output stage (50V, 5A)]
//           Rack#2B-20 DR_ZF (EL7047) [EL7047 1Ch. Stepper motor output stage (50V, 5A)]
//           Rack#2B-21 EtherCAT Extension (EK1110) [EK1110 EtherCAT extension]
//         Rack#2D LinearGaugeAmp (SC-HG1-ETC) [SC-HG1-ETC]
// variable links:
//   CX2020 (EtherCAT) <-> CX2020 (EtherCAT)/Term 1 (EK1200)/Term 2 (EK1122)/Rack#1A-01 Coupler (EK1100)/Rack#1A-02 SFIN (EL1918)
//     Term 1 (EK1200)/Term 2 (EK1122)/BOX-01 Coupler (EK1100)/BOX-02 SFIN(EL1904)/Module 1 (FSOES)/RxPDO/FSOE <-> ConnectionInputs/Message_4 TxPDO
//     Term 1 (EK1200)/Term 2 (EK1122)/BOX-01 Coupler (EK1100)/BOX-02 SFIN(EL1904)/Module 1 (FSOES)/TxPDO/FSOE <-> ConnectionOutputs/Message_4 RxPDO
//   CX2020 (EtherCAT) <-> CX2020 (EtherCAT)/Term 1 (EK1200)/Term 2 (EK1122)/Rack#1A-01 Coupler (EK1100)/Rack#1A-03 SFOUT(EL2912)
//     Term 1 (EK1200)/Term 2 (EK1122)/Rack#1A-01 Coupler (EK1100)/Rack#1A-02 SFIN (EL1918)/ConnectionInputs/Message_3 TxPDO <-> Module 1 (FSOE)/FSoE Outputs/FSOE
//     Term 1 (EK1200)/Term 2 (EK1122)/Rack#1A-01 Coupler (EK1100)/Rack#1A-02 SFIN (EL1918)/ConnectionOutputs/Message_3 RxPDO <-> Module 1 (FSOE)/FSoE Inputs/FSOE
//   CX2020 (EtherCAT) <-> CX2020 (EtherCAT)/Term 1 (EK1200)/Term 2 (EK1122)/Rack#2B-01 Coupler (EK1100)/Rack#2B-06 SFIN (EL1918)
//     Term 1 (EK1200)/Term 2 (EK1122)/Rack#1A-01 Coupler (EK1100)/Rack#1A-02 SFIN (EL1918)/ConnectionInputs/Message_6 TxPDO <-> Module 1 (FSOE)/FSoE Outputs/FSOE
//     Term 1 (EK1200)/Term 2 (EK1122)/Rack#1A-01 Coupler (EK1100)/Rack#1A-02 SFIN (EL1918)/ConnectionOutputs/Message_6 RxPDO <-> Module 1 (FSOE)/FSoE Inputs/FSOE
//   NC-Task 1 SAF/Axes/RxG <-> CX2020 (EtherCAT)/Term 1 (EK1200)/Term 2 (EK1122)/Rack#2A-01 Coupler (EK1100)/Rack#2A-08 DR_RxG (EL7041-0052)
//     Drive/Inputs/In/nState1 @bit 3 <-> STM Status/Status/Error
//     Drive/Inputs/In/nState1 @bit 5 <-> STM Status/Status/Moving negative
//     Drive/Inputs/In/nState1 @bit 4 <-> STM Status/Status/Moving positive
//     Drive/Inputs/In/nState1 @bit 1 <-> STM Status/Status/Ready
//     Drive/Inputs/In/nState1 <-> STM Status/Status/Ready to enable
//     Drive/Inputs/In/nState1 @bit 6 <-> STM Status/Status/Torque reduced
//     Drive/Inputs/In/nState1 @bit 2 <-> STM Status/Status/Warning
//     Drive/Inputs/In/nState2 @bit 3 <-> STM Status/Status/Digital input 1
//     Drive/Inputs/In/nState2 @bit 4 <-> STM Status/Status/Digital input 2
//     Drive/Inputs/In/nState2 @bit 5 <-> STM Status/Status/Sync error
//     Drive/Inputs/In/nState2 @bit 7 <-> STM Status/Status/TxPDO Toggle
//     Drive/Inputs/In/nState4 @bit 1 <-> WcState/InputToggle
//     Drive/Inputs/In/nState4 <-> WcState/WcState
//     Drive/Outputs/Out/nCtrl1 <-> STM Control/Control/Enable
//     Drive/Outputs/Out/nCtrl1 @bit 2 <-> STM Control/Control/Reduce torque
//     Drive/Outputs/Out/nCtrl1 @bit 1 <-> STM Control/Control/Reset
//     Drive/Outputs/Out/nDataOut2[0] <-> STM Velocity/Velocity
//   NC-Task 1 SAF/Axes/RxG <-> CX2020 (EtherCAT)/Term 1 (EK1200)/Term 2 (EK1122)/Rack#2B-01 Coupler (EK1100)/Rack#2B-09 ENC_RxG_XG (EL5042)
//     Enc/Inputs/In/nDataIn1 <-> FB Inputs Channel 1 compact/Position
//     Enc/Inputs/In/nDcInputTime <-> InfoData/DcInputShift
//     Enc/Inputs/In/nState1 @bit 1 <-> FB Inputs Channel 1 compact/Status/Error
//     Enc/Inputs/In/nState1 @bit 2 <-> FB Inputs Channel 1 compact/Status/Ready
//     Enc/Inputs/In/nState1 <-> FB Inputs Channel 1 compact/Status/Warning
//     Enc/Inputs/In/nState2 @bit 4 <-> FB Inputs Channel 1 compact/Status/Diag
//     Enc/Inputs/In/nState2 @bit 6 <-> FB Inputs Channel 1 compact/Status/Input cycle counter
//     Enc/Inputs/In/nState2 @bit 5 <-> FB Inputs Channel 1 compact/Status/TxPDO State
//     Enc/Inputs/In/nState4 @bit 1 <-> WcState/InputToggle
//     Enc/Inputs/In/nState4 <-> WcState/WcState
//   NC-Task 1 SAF/Axes/RyDC <-> CX2020 (EtherCAT)/Term 1 (EK1200)/Term 2 (EK1122)/BOX-01 Coupler (EK1100)/BOX-05 ENC_XDC_RyDC (EL5042)
//     Enc/Inputs/In/nComState @bit 1 <-> WcState/InputToggle
//     Enc/Inputs/In/nComState <-> WcState/WcState
//     Enc/Inputs/In/nDataIn1 <-> FB Inputs Channel 2/Position
//     Enc/Inputs/In/nState1 @bit 12 <-> FB Inputs Channel 2/Status/Diag
//     Enc/Inputs/In/nState1 @bit 1 <-> FB Inputs Channel 2/Status/Error
//     Enc/Inputs/In/nState1 @bit 14 <-> FB Inputs Channel 2/Status/Input cycle counter
//     Enc/Inputs/In/nState1 @bit 2 <-> FB Inputs Channel 2/Status/Ready
//     Enc/Inputs/In/nState1 @bit 13 <-> FB Inputs Channel 2/Status/TxPDO State
//     Enc/Inputs/In/nState1 <-> FB Inputs Channel 2/Status/Warning
//   NC-Task 1 SAF/Axes/RyDC <-> CX2020 (EtherCAT)/Term 1 (EK1200)/Term 2 (EK1122)/BOX-01 Coupler (EK1100)/BOX-15 DR_RyDC (EL7041-0052)
//     Drive/Inputs/In/nState1 @bit 3 <-> STM Status/Status/Error
//     Drive/Inputs/In/nState1 @bit 5 <-> STM Status/Status/Moving negative
//     Drive/Inputs/In/nState1 @bit 4 <-> STM Status/Status/Moving positive
//     Drive/Inputs/In/nState1 @bit 1 <-> STM Status/Status/Ready
//     Drive/Inputs/In/nState1 <-> STM Status/Status/Ready to enable
//     Drive/Inputs/In/nState1 @bit 6 <-> STM Status/Status/Torque reduced
//     Drive/Inputs/In/nState1 @bit 2 <-> STM Status/Status/Warning
//     Drive/Inputs/In/nState2 @bit 3 <-> STM Status/Status/Digital input 1
//     Drive/Inputs/In/nState2 @bit 4 <-> STM Status/Status/Digital input 2
//     Drive/Inputs/In/nState2 @bit 5 <-> STM Status/Status/Sync error
//     Drive/Inputs/In/nState2 @bit 7 <-> STM Status/Status/TxPDO Toggle
//     Drive/Inputs/In/nState4 @bit 1 <-> WcState/InputToggle
//     Drive/Inputs/In/nState4 <-> WcState/WcState
//     Drive/Outputs/Out/nCtrl1 <-> STM Control/Control/Enable
//     Drive/Outputs/Out/nCtrl1 @bit 2 <-> STM Control/Control/Reduce torque
//     Drive/Outputs/Out/nCtrl1 @bit 1 <-> STM Control/Control/Reset
//     Drive/Outputs/Out/nDataOut2[0] <-> STM Velocity/Velocity
//   NC-Task 1 SAF/Axes/RzPM <-> CX2020 (EtherCAT)/Term 1 (EK1200)/Term 2 (EK1122)/Rack#2A-01 Coupler (EK1100)/Rack#2A-16 DR_RzPM (EL7041-0052)
//     Drive/Inputs/In/nState1 @bit 3 <-> STM Status/Status/Error
//     Drive/Inputs/In/nState1 @bit 5 <-> STM Status/Status/Moving negative
//     Drive/Inputs/In/nState1 @bit 4 <-> STM Status/Status/Moving positive
//     Drive/Inputs/In/nState1 @bit 1 <-> STM Status/Status/Ready
//     Drive/Inputs/In/nState1 <-> STM Status/Status/Ready to enable
//     Drive/Inputs/In/nState1 @bit 6 <-> STM Status/Status/Torque reduced
//     Drive/Inputs/In/nState1 @bit 2 <-> STM Status/Status/Warning
//     Drive/Inputs/In/nState2 @bit 3 <-> STM Status/Status/Digital input 1
//     Drive/Inputs/In/nState2 @bit 4 <-> STM Status/Status/Digital input 2
//     Drive/Inputs/In/nState2 @bit 5 <-> STM Status/Status/Sync error
//     Drive/Inputs/In/nState2 @bit 7 <-> STM Status/Status/TxPDO Toggle
//     Drive/Inputs/In/nState4 @bit 1 <-> WcState/InputToggle
//     Drive/Inputs/In/nState4 <-> WcState/WcState
//     Drive/Outputs/Out/nCtrl1 <-> STM Control/Control/Enable
//     Drive/Outputs/Out/nCtrl1 @bit 2 <-> STM Control/Control/Reduce torque
//     Drive/Outputs/Out/nCtrl1 @bit 1 <-> STM Control/Control/Reset
//     Drive/Outputs/Out/nDataOut2[0] <-> STM Velocity/Velocity
//   NC-Task 1 SAF/Axes/RzPM <-> CX2020 (EtherCAT)/Term 1 (EK1200)/Term 2 (EK1122)/Rack#2B-01 Coupler (EK1100)/Rack#2B-12 ENC_X2PM_RzPM (EL5042)
//     Enc/Inputs/In/nComState @bit 1 <-> WcState/InputToggle
//     Enc/Inputs/In/nComState <-> WcState/WcState
//     Enc/Inputs/In/nDataIn1 <-> FB Inputs Channel 2/Position
//     Enc/Inputs/In/nDcInputTime <-> InfoData/DcInputShift
//     Enc/Inputs/In/nState1 @bit 12 <-> FB Inputs Channel 2/Status/Diag
//     Enc/Inputs/In/nState1 @bit 1 <-> FB Inputs Channel 2/Status/Error
//     Enc/Inputs/In/nState1 @bit 14 <-> FB Inputs Channel 2/Status/Input cycle counter
//     Enc/Inputs/In/nState1 @bit 2 <-> FB Inputs Channel 2/Status/Ready
//     Enc/Inputs/In/nState1 @bit 13 <-> FB Inputs Channel 2/Status/TxPDO State
//     Enc/Inputs/In/nState1 <-> FB Inputs Channel 2/Status/Warning
//   NC-Task 1 SAF/Axes/ServoDrive <-> CX2020 (EtherCAT)/Term 1 (EK1200)/Term 2 (EK1122)/Rack#1C_ServoDR (NCR-HD Series)
//     Drive/Inputs/In/nDataIn1 <-> 260th transmit PDO Mapping/Following error actual value
//     Drive/Inputs/In/nDataIn3[0] <-> 260th transmit PDO Mapping/Torque actual value
//     Drive/Inputs/In/nDcOutputTime <-> InfoData/DcOutputShift
//     Drive/Inputs/In/nState1 <-> 260th transmit PDO Mapping/Statusword
//     Drive/Inputs/In/nState2 <-> 260th transmit PDO Mapping/Statusword @bit 8
//     Drive/Inputs/In/nState4 @bit 1 <-> WcState/InputToggle
//     Drive/Inputs/In/nState4 <-> WcState/WcState
//     Drive/Inputs/In/nState5 <-> 260th transmit PDO Mapping/Modes of operation display
//     Drive/Outputs/Out/nCtrl1 <-> 260th receive PDO Mapping/Controlword
//     Drive/Outputs/Out/nCtrl2 <-> 260th receive PDO Mapping/Controlword @bit 8
//     Drive/Outputs/Out/nCtrl5 <-> 260th receive PDO Mapping/Modes of operation
//     Drive/Outputs/Out/nDataOut1 <-> 260th receive PDO Mapping/Target position
//     Drive/Outputs/Out/nDataOut2 <-> 260th receive PDO Mapping/Target velocity
//     Enc/Inputs/In/nDataIn1 <-> 260th transmit PDO Mapping/Position actual value
//     Enc/Inputs/In/nDataIn3 <-> 260th transmit PDO Mapping/Touch probe pos1 pos value
//     Enc/Inputs/In/nDataIn5 <-> 260th transmit PDO Mapping/Touch probe pos2 pos value
//     Enc/Inputs/In/nDcInputTime <-> InfoData/DcInputShift
//     Enc/Inputs/In/nState4 @bit 1 <-> WcState/InputToggle
//     Enc/Inputs/In/nState4 <-> WcState/WcState
//     Enc/Inputs/In/nState5 <-> 260th transmit PDO Mapping/Touch probe status
//     Enc/Inputs/In/nState6 <-> 260th transmit PDO Mapping/Touch probe status @bit 8
//     Enc/Outputs/Out/nCtrl5 <-> 260th receive PDO Mapping/Touch probe function
//     Enc/Outputs/Out/nCtrl6 <-> 260th receive PDO Mapping/Touch probe function @bit 8
//   NC-Task 1 SAF/Axes/Stepper <-> CX2020 (EtherCAT)/Term 1 (EK1200)/Term 2 (EK1122)/Rack#1A-01 Coupler (EK1100)/Rack#1A-04 DR_2Th (EL7047)
//     Drive/Inputs/In/nState1 @bit 3 <-> STM Status/Status/Error
//     Drive/Inputs/In/nState1 @bit 7 <-> STM Status/Status/Motor stall
//     Drive/Inputs/In/nState1 @bit 5 <-> STM Status/Status/Moving negative
//     Drive/Inputs/In/nState1 @bit 4 <-> STM Status/Status/Moving positive
//     Drive/Inputs/In/nState1 @bit 1 <-> STM Status/Status/Ready
//     Drive/Inputs/In/nState1 <-> STM Status/Status/Ready to enable
//     Drive/Inputs/In/nState1 @bit 6 <-> STM Status/Status/Torque reduced
//     Drive/Inputs/In/nState1 @bit 2 <-> STM Status/Status/Warning
//     Drive/Inputs/In/nState2 @bit 3 <-> STM Status/Status/Digital input 1
//     Drive/Inputs/In/nState2 @bit 4 <-> STM Status/Status/Digital input 2
//     Drive/Inputs/In/nState2 @bit 5 <-> STM Status/Status/Sync error
//     Drive/Inputs/In/nState2 @bit 7 <-> STM Status/Status/TxPDO Toggle
//     Drive/Inputs/In/nState4 @bit 1 <-> WcState/InputToggle
//     Drive/Inputs/In/nState4 <-> WcState/WcState
//     Drive/Outputs/Out/nCtrl1 <-> STM Control/Control/Enable
//     Drive/Outputs/Out/nCtrl1 @bit 2 <-> STM Control/Control/Reduce torque
//     Drive/Outputs/Out/nCtrl1 @bit 1 <-> STM Control/Control/Reset
//     Drive/Outputs/Out/nCtrl2 @bit 3 <-> STM Control/Control/Digital output 1
//     Drive/Outputs/Out/nDataOut2[0] <-> STM Velocity/Velocity
//   NC-Task 1 SAF/Axes/Stepper <-> CX2020 (EtherCAT)/Term 1 (EK1200)/Term 2 (EK1122)/Rack#1A-01 Coupler (EK1100)/Rack#1A-06 ENC_2Th (EL5042)
//     Enc/Inputs/In/nComState @bit 1 <-> WcState/InputToggle
//     Enc/Inputs/In/nComState <-> WcState/WcState
//     Enc/Inputs/In/nDataIn1 <-> FB Inputs Channel 1/Position
//     Enc/Inputs/In/nDcInputTime <-> InfoData/DcInputShift
//     Enc/Inputs/In/nState1 @bit 12 <-> FB Inputs Channel 1/Status/Diag
//     Enc/Inputs/In/nState1 @bit 1 <-> FB Inputs Channel 1/Status/Error
//     Enc/Inputs/In/nState1 @bit 14 <-> FB Inputs Channel 1/Status/Input cycle counter
//     Enc/Inputs/In/nState1 @bit 2 <-> FB Inputs Channel 1/Status/Ready
//     Enc/Inputs/In/nState1 @bit 13 <-> FB Inputs Channel 1/Status/TxPDO State
//     Enc/Inputs/In/nState1 <-> FB Inputs Channel 1/Status/Warning
//   NC-Task 1 SAF/Axes/XDC <-> CX2020 (EtherCAT)/Term 1 (EK1200)/Term 2 (EK1122)/BOX-01 Coupler (EK1100)/BOX-05 ENC_XDC_RyDC (EL5042)
//     Enc/Inputs/In/nComState @bit 1 <-> WcState/InputToggle
//     Enc/Inputs/In/nComState <-> WcState/WcState
//     Enc/Inputs/In/nDataIn1 <-> FB Inputs Channel 1/Position
//     Enc/Inputs/In/nState1 @bit 12 <-> FB Inputs Channel 1/Status/Diag
//     Enc/Inputs/In/nState1 @bit 1 <-> FB Inputs Channel 1/Status/Error
//     Enc/Inputs/In/nState1 @bit 14 <-> FB Inputs Channel 1/Status/Input cycle counter
//     Enc/Inputs/In/nState1 @bit 2 <-> FB Inputs Channel 1/Status/Ready
//     Enc/Inputs/In/nState1 @bit 13 <-> FB Inputs Channel 1/Status/TxPDO State
//     Enc/Inputs/In/nState1 <-> FB Inputs Channel 1/Status/Warning
//   NC-Task 1 SAF/Axes/XDC <-> CX2020 (EtherCAT)/Term 1 (EK1200)/Term 2 (EK1122)/BOX-01 Coupler (EK1100)/BOX-14 DR_XDC (EL7041-0052)
//     Drive/Inputs/In/nState1 @bit 3 <-> STM Status/Status/Error
//     Drive/Inputs/In/nState1 @bit 5 <-> STM Status/Status/Moving negative
//     Drive/Inputs/In/nState1 @bit 4 <-> STM Status/Status/Moving positive
//     Drive/Inputs/In/nState1 @bit 1 <-> STM Status/Status/Ready
//     Drive/Inputs/In/nState1 <-> STM Status/Status/Ready to enable
//     Drive/Inputs/In/nState1 @bit 6 <-> STM Status/Status/Torque reduced
//     Drive/Inputs/In/nState1 @bit 2 <-> STM Status/Status/Warning
//     Drive/Inputs/In/nState2 @bit 3 <-> STM Status/Status/Digital input 1
//     Drive/Inputs/In/nState2 @bit 4 <-> STM Status/Status/Digital input 2
//     Drive/Inputs/In/nState2 @bit 5 <-> STM Status/Status/Sync error
//     Drive/Inputs/In/nState2 @bit 7 <-> STM Status/Status/TxPDO Toggle
//     Drive/Inputs/In/nState4 @bit 1 <-> WcState/InputToggle
//     Drive/Inputs/In/nState4 <-> WcState/WcState
//     Drive/Outputs/Out/nCtrl1 <-> STM Control/Control/Enable
//     Drive/Outputs/Out/nCtrl1 @bit 2 <-> STM Control/Control/Reduce torque
//     Drive/Outputs/Out/nCtrl1 @bit 1 <-> STM Control/Control/Reset
//     Drive/Outputs/Out/nDataOut2[0] <-> STM Velocity/Velocity
//   NC-Task 1 SAF/Axes/XG <-> CX2020 (EtherCAT)/Term 1 (EK1200)/Term 2 (EK1122)/Rack#2A-01 Coupler (EK1100)/Rack#2A-09 DR_XG (EL7041-0052)
//     Drive/Inputs/In/nState1 @bit 3 <-> STM Status/Status/Error
//     Drive/Inputs/In/nState1 @bit 5 <-> STM Status/Status/Moving negative
//     Drive/Inputs/In/nState1 @bit 4 <-> STM Status/Status/Moving positive
//     Drive/Inputs/In/nState1 @bit 1 <-> STM Status/Status/Ready
//     Drive/Inputs/In/nState1 <-> STM Status/Status/Ready to enable
//     Drive/Inputs/In/nState1 @bit 6 <-> STM Status/Status/Torque reduced
//     Drive/Inputs/In/nState1 @bit 2 <-> STM Status/Status/Warning
//     Drive/Inputs/In/nState2 @bit 3 <-> STM Status/Status/Digital input 1
//     Drive/Inputs/In/nState2 @bit 4 <-> STM Status/Status/Digital input 2
//     Drive/Inputs/In/nState2 @bit 5 <-> STM Status/Status/Sync error
//     Drive/Inputs/In/nState2 @bit 7 <-> STM Status/Status/TxPDO Toggle
//     Drive/Inputs/In/nState4 @bit 1 <-> WcState/InputToggle
//     Drive/Inputs/In/nState4 <-> WcState/WcState
//     Drive/Outputs/Out/nCtrl1 <-> STM Control/Control/Enable
//     Drive/Outputs/Out/nCtrl1 @bit 2 <-> STM Control/Control/Reduce torque
//     Drive/Outputs/Out/nCtrl1 @bit 1 <-> STM Control/Control/Reset
//     Drive/Outputs/Out/nDataOut2[0] <-> STM Velocity/Velocity
//   NC-Task 1 SAF/Axes/XG <-> CX2020 (EtherCAT)/Term 1 (EK1200)/Term 2 (EK1122)/Rack#2B-01 Coupler (EK1100)/Rack#2B-09 ENC_RxG_XG (EL5042)
//     Enc/Inputs/In/nComState @bit 1 <-> WcState/InputToggle
//     Enc/Inputs/In/nComState <-> WcState/WcState
//     Enc/Inputs/In/nDataIn1 <-> FB Inputs Channel 2/Position
//     Enc/Inputs/In/nDcInputTime <-> InfoData/DcInputShift
//     Enc/Inputs/In/nState1 @bit 12 <-> FB Inputs Channel 2/Status/Diag
//     Enc/Inputs/In/nState1 @bit 1 <-> FB Inputs Channel 2/Status/Error
//     Enc/Inputs/In/nState1 @bit 14 <-> FB Inputs Channel 2/Status/Input cycle counter
//     Enc/Inputs/In/nState1 @bit 2 <-> FB Inputs Channel 2/Status/Ready
//     Enc/Inputs/In/nState1 @bit 13 <-> FB Inputs Channel 2/Status/TxPDO State
//     Enc/Inputs/In/nState1 <-> FB Inputs Channel 2/Status/Warning
//   NC-Task 1 SAF/Axes/XPM1 <-> CX2020 (EtherCAT)/Term 1 (EK1200)/Term 2 (EK1122)/Rack#2A-01 Coupler (EK1100)/Rack#2A-14 DR_XPM1 (EL7041-0052)
//     Drive/Inputs/In/nDcOutputTime <-> InfoData/DcOutputShift
//     Drive/Inputs/In/nState1 @bit 3 <-> STM Status/Status/Error
//     Drive/Inputs/In/nState1 @bit 5 <-> STM Status/Status/Moving negative
//     Drive/Inputs/In/nState1 @bit 4 <-> STM Status/Status/Moving positive
//     Drive/Inputs/In/nState1 @bit 1 <-> STM Status/Status/Ready
//     Drive/Inputs/In/nState1 <-> STM Status/Status/Ready to enable
//     Drive/Inputs/In/nState1 @bit 6 <-> STM Status/Status/Torque reduced
//     Drive/Inputs/In/nState1 @bit 2 <-> STM Status/Status/Warning
//     Drive/Inputs/In/nState2 @bit 3 <-> STM Status/Status/Digital input 1
//     Drive/Inputs/In/nState2 @bit 4 <-> STM Status/Status/Digital input 2
//     Drive/Inputs/In/nState2 @bit 5 <-> STM Status/Status/Sync error
//     Drive/Inputs/In/nState2 @bit 7 <-> STM Status/Status/TxPDO Toggle
//     Drive/Inputs/In/nState4 @bit 1 <-> WcState/InputToggle
//     Drive/Inputs/In/nState4 <-> WcState/WcState
//     Drive/Outputs/Out/nCtrl1 <-> STM Control/Control/Enable
//     Drive/Outputs/Out/nCtrl1 @bit 2 <-> STM Control/Control/Reduce torque
//     Drive/Outputs/Out/nCtrl1 @bit 1 <-> STM Control/Control/Reset
//     Drive/Outputs/Out/nDataOut2[0] <-> STM Velocity/Velocity
//   NC-Task 1 SAF/Axes/XPM1 <-> CX2020 (EtherCAT)/Term 1 (EK1200)/Term 2 (EK1122)/Rack#2B-01 Coupler (EK1100)/Rack#2B-11 ENC_YG3_X1PM (EL5042)
//     Enc/Inputs/In/nComState @bit 1 <-> WcState/InputToggle
//     Enc/Inputs/In/nComState <-> WcState/WcState
//     Enc/Inputs/In/nDataIn1 <-> FB Inputs Channel 2/Position
//     Enc/Inputs/In/nDcInputTime <-> InfoData/DcInputShift
//     Enc/Inputs/In/nState1 @bit 12 <-> FB Inputs Channel 2/Status/Diag
//     Enc/Inputs/In/nState1 @bit 1 <-> FB Inputs Channel 2/Status/Error
//     Enc/Inputs/In/nState1 @bit 14 <-> FB Inputs Channel 2/Status/Input cycle counter
//     Enc/Inputs/In/nState1 @bit 2 <-> FB Inputs Channel 2/Status/Ready
//     Enc/Inputs/In/nState1 @bit 13 <-> FB Inputs Channel 2/Status/TxPDO State
//     Enc/Inputs/In/nState1 <-> FB Inputs Channel 2/Status/Warning
//   NC-Task 1 SAF/Axes/XPM2 <-> CX2020 (EtherCAT)/Term 1 (EK1200)/Term 2 (EK1122)/Rack#2A-01 Coupler (EK1100)/Rack#2A-15 DR_XPM2 (EL7041-0052)
//     Drive/Inputs/In/nState1 @bit 3 <-> STM Status/Status/Error
//     Drive/Inputs/In/nState1 @bit 5 <-> STM Status/Status/Moving negative
//     Drive/Inputs/In/nState1 @bit 4 <-> STM Status/Status/Moving positive
//     Drive/Inputs/In/nState1 @bit 1 <-> STM Status/Status/Ready
//     Drive/Inputs/In/nState1 <-> STM Status/Status/Ready to enable
//     Drive/Inputs/In/nState1 @bit 6 <-> STM Status/Status/Torque reduced
//     Drive/Inputs/In/nState1 @bit 2 <-> STM Status/Status/Warning
//     Drive/Inputs/In/nState2 @bit 3 <-> STM Status/Status/Digital input 1
//     Drive/Inputs/In/nState2 @bit 4 <-> STM Status/Status/Digital input 2
//     Drive/Inputs/In/nState2 @bit 5 <-> STM Status/Status/Sync error
//     Drive/Inputs/In/nState2 @bit 7 <-> STM Status/Status/TxPDO Toggle
//     Drive/Inputs/In/nState4 @bit 1 <-> WcState/InputToggle
//     Drive/Inputs/In/nState4 <-> WcState/WcState
//     Drive/Outputs/Out/nCtrl1 <-> STM Control/Control/Enable
//     Drive/Outputs/Out/nCtrl1 @bit 2 <-> STM Control/Control/Reduce torque
//     Drive/Outputs/Out/nCtrl1 @bit 1 <-> STM Control/Control/Reset
//     Drive/Outputs/Out/nDataOut2[0] <-> STM Velocity/Velocity
//   NC-Task 1 SAF/Axes/XPM2 <-> CX2020 (EtherCAT)/Term 1 (EK1200)/Term 2 (EK1122)/Rack#2B-01 Coupler (EK1100)/Rack#2B-12 ENC_X2PM_RzPM (EL5042)
//     Enc/Inputs/In/nComState @bit 1 <-> WcState/InputToggle
//     Enc/Inputs/In/nComState <-> WcState/WcState
//     Enc/Inputs/In/nDataIn1 <-> FB Inputs Channel 1/Position
//     Enc/Inputs/In/nDcInputTime <-> InfoData/DcInputShift
//     Enc/Inputs/In/nState1 @bit 12 <-> FB Inputs Channel 1/Status/Diag
//     Enc/Inputs/In/nState1 @bit 1 <-> FB Inputs Channel 1/Status/Error
//     Enc/Inputs/In/nState1 @bit 14 <-> FB Inputs Channel 1/Status/Input cycle counter
//     Enc/Inputs/In/nState1 @bit 2 <-> FB Inputs Channel 1/Status/Ready
//     Enc/Inputs/In/nState1 @bit 13 <-> FB Inputs Channel 1/Status/TxPDO State
//     Enc/Inputs/In/nState1 <-> FB Inputs Channel 1/Status/Warning
//   NC-Task 1 SAF/Axes/XS1 <-> CX2020 (EtherCAT)/Term 1 (EK1200)/Term 2 (EK1122)/Rack#2A-01 Coupler (EK1100)/Rack#2A-03 DR_XS1 (EL7041-0052)
//     Drive/Inputs/In/nDcOutputTime <-> InfoData/DcOutputShift
//     Drive/Inputs/In/nState1 @bit 3 <-> STM Status/Status/Error
//     Drive/Inputs/In/nState1 @bit 5 <-> STM Status/Status/Moving negative
//     Drive/Inputs/In/nState1 @bit 4 <-> STM Status/Status/Moving positive
//     Drive/Inputs/In/nState1 @bit 1 <-> STM Status/Status/Ready
//     Drive/Inputs/In/nState1 <-> STM Status/Status/Ready to enable
//     Drive/Inputs/In/nState1 @bit 6 <-> STM Status/Status/Torque reduced
//     Drive/Inputs/In/nState1 @bit 2 <-> STM Status/Status/Warning
//     Drive/Inputs/In/nState2 @bit 3 <-> STM Status/Status/Digital input 1
//     Drive/Inputs/In/nState2 @bit 4 <-> STM Status/Status/Digital input 2
//     Drive/Inputs/In/nState2 @bit 5 <-> STM Status/Status/Sync error
//     Drive/Inputs/In/nState2 @bit 7 <-> STM Status/Status/TxPDO Toggle
//     Drive/Inputs/In/nState4 @bit 1 <-> WcState/InputToggle
//     Drive/Inputs/In/nState4 <-> WcState/WcState
//     Drive/Outputs/Out/nCtrl1 <-> STM Control/Control/Enable
//     Drive/Outputs/Out/nCtrl1 @bit 2 <-> STM Control/Control/Reduce torque
//     Drive/Outputs/Out/nCtrl1 @bit 1 <-> STM Control/Control/Reset
//     Drive/Outputs/Out/nDataOut2[0] <-> STM Velocity/Velocity
//   NC-Task 1 SAF/Axes/XS1 <-> CX2020 (EtherCAT)/Term 1 (EK1200)/Term 2 (EK1122)/Rack#2B-01 Coupler (EK1100)/Rack#2B-07 ENC_X1_X2 (EL5042)
//     Enc/Inputs/In/nComState @bit 1 <-> WcState/InputToggle
//     Enc/Inputs/In/nComState <-> WcState/WcState
//     Enc/Inputs/In/nDataIn1 <-> FB Inputs Channel 1/Position
//     Enc/Inputs/In/nDcInputTime <-> InfoData/DcInputShift
//     Enc/Inputs/In/nState1 @bit 12 <-> FB Inputs Channel 1/Status/Diag
//     Enc/Inputs/In/nState1 @bit 1 <-> FB Inputs Channel 1/Status/Error
//     Enc/Inputs/In/nState1 @bit 14 <-> FB Inputs Channel 1/Status/Input cycle counter
//     Enc/Inputs/In/nState1 @bit 2 <-> FB Inputs Channel 1/Status/Ready
//     Enc/Inputs/In/nState1 @bit 13 <-> FB Inputs Channel 1/Status/TxPDO State
//     Enc/Inputs/In/nState1 <-> FB Inputs Channel 1/Status/Warning
//   NC-Task 1 SAF/Axes/XS2 <-> CX2020 (EtherCAT)/Term 1 (EK1200)/Term 2 (EK1122)/Rack#2A-01 Coupler (EK1100)/Rack#2A-04 DR_XS2 (EL7041-0052)
//     Drive/Inputs/In/nDcOutputTime <-> InfoData/DcOutputShift
//     Drive/Inputs/In/nState1 @bit 3 <-> STM Status/Status/Error
//     Drive/Inputs/In/nState1 @bit 5 <-> STM Status/Status/Moving negative
//     Drive/Inputs/In/nState1 @bit 4 <-> STM Status/Status/Moving positive
//     Drive/Inputs/In/nState1 @bit 1 <-> STM Status/Status/Ready
//     Drive/Inputs/In/nState1 <-> STM Status/Status/Ready to enable
//     Drive/Inputs/In/nState1 @bit 6 <-> STM Status/Status/Torque reduced
//     Drive/Inputs/In/nState1 @bit 2 <-> STM Status/Status/Warning
//     Drive/Inputs/In/nState2 @bit 3 <-> STM Status/Status/Digital input 1
//     Drive/Inputs/In/nState2 @bit 4 <-> STM Status/Status/Digital input 2
//     Drive/Inputs/In/nState2 @bit 5 <-> STM Status/Status/Sync error
//     Drive/Inputs/In/nState2 @bit 7 <-> STM Status/Status/TxPDO Toggle
//     Drive/Inputs/In/nState4 @bit 1 <-> WcState/InputToggle
//     Drive/Inputs/In/nState4 <-> WcState/WcState
//     Drive/Outputs/Out/nCtrl1 <-> STM Control/Control/Enable
//     Drive/Outputs/Out/nCtrl1 @bit 2 <-> STM Control/Control/Reduce torque
//     Drive/Outputs/Out/nCtrl1 @bit 1 <-> STM Control/Control/Reset
//     Drive/Outputs/Out/nDataOut2[0] <-> STM Velocity/Velocity
//   NC-Task 1 SAF/Axes/XS2 <-> CX2020 (EtherCAT)/Term 1 (EK1200)/Term 2 (EK1122)/Rack#2B-01 Coupler (EK1100)/Rack#2B-07 ENC_X1_X2 (EL5042)
//     Enc/Inputs/In/nComState @bit 1 <-> WcState/InputToggle
//     Enc/Inputs/In/nComState <-> WcState/WcState
//     Enc/Inputs/In/nDataIn1 <-> FB Inputs Channel 2/Position
//     Enc/Inputs/In/nDcInputTime <-> InfoData/DcInputShift
//     Enc/Inputs/In/nState1 @bit 12 <-> FB Inputs Channel 2/Status/Diag
//     Enc/Inputs/In/nState1 @bit 1 <-> FB Inputs Channel 2/Status/Error
//     Enc/Inputs/In/nState1 @bit 14 <-> FB Inputs Channel 2/Status/Input cycle counter
//     Enc/Inputs/In/nState1 @bit 2 <-> FB Inputs Channel 2/Status/Ready
//     Enc/Inputs/In/nState1 @bit 13 <-> FB Inputs Channel 2/Status/TxPDO State
//     Enc/Inputs/In/nState1 <-> FB Inputs Channel 2/Status/Warning
//   NC-Task 1 SAF/Axes/XSDC1 <-> CX2020 (EtherCAT)/Term 1 (EK1200)/Term 2 (EK1122)/BOX-01 Coupler (EK1100)/BOX-03 ENC_X1_X2 (EL5042)
//     Enc/Inputs/In/nComState @bit 1 <-> WcState/InputToggle
//     Enc/Inputs/In/nComState <-> WcState/WcState
//     Enc/Inputs/In/nDataIn1 <-> FB Inputs Channel 1/Position
//     Enc/Inputs/In/nDcInputTime <-> InfoData/DcInputShift
//     Enc/Inputs/In/nState1 @bit 12 <-> FB Inputs Channel 1/Status/Diag
//     Enc/Inputs/In/nState1 @bit 1 <-> FB Inputs Channel 1/Status/Error
//     Enc/Inputs/In/nState1 @bit 14 <-> FB Inputs Channel 1/Status/Input cycle counter
//     Enc/Inputs/In/nState1 @bit 2 <-> FB Inputs Channel 1/Status/Ready
//     Enc/Inputs/In/nState1 @bit 13 <-> FB Inputs Channel 1/Status/TxPDO State
//     Enc/Inputs/In/nState1 <-> FB Inputs Channel 1/Status/Warning
//   NC-Task 1 SAF/Axes/XSDC1 <-> CX2020 (EtherCAT)/Term 1 (EK1200)/Term 2 (EK1122)/BOX-01 Coupler (EK1100)/BOX-09 DR_XSDC1 (EL7041-0052)
//     Drive/Inputs/In/nState1 @bit 3 <-> STM Status/Status/Error
//     Drive/Inputs/In/nState1 @bit 5 <-> STM Status/Status/Moving negative
//     Drive/Inputs/In/nState1 @bit 4 <-> STM Status/Status/Moving positive
//     Drive/Inputs/In/nState1 @bit 1 <-> STM Status/Status/Ready
//     Drive/Inputs/In/nState1 <-> STM Status/Status/Ready to enable
//     Drive/Inputs/In/nState1 @bit 6 <-> STM Status/Status/Torque reduced
//     Drive/Inputs/In/nState1 @bit 2 <-> STM Status/Status/Warning
//     Drive/Inputs/In/nState2 @bit 3 <-> STM Status/Status/Digital input 1
//     Drive/Inputs/In/nState2 @bit 4 <-> STM Status/Status/Digital input 2
//     Drive/Inputs/In/nState2 @bit 5 <-> STM Status/Status/Sync error
//     Drive/Inputs/In/nState2 @bit 7 <-> STM Status/Status/TxPDO Toggle
//     Drive/Inputs/In/nState4 @bit 1 <-> WcState/InputToggle
//     Drive/Inputs/In/nState4 <-> WcState/WcState
//     Drive/Outputs/Out/nCtrl1 <-> STM Control/Control/Enable
//     Drive/Outputs/Out/nCtrl1 @bit 2 <-> STM Control/Control/Reduce torque
//     Drive/Outputs/Out/nCtrl1 @bit 1 <-> STM Control/Control/Reset
//     Drive/Outputs/Out/nDataOut2[0] <-> STM Velocity/Velocity
//   NC-Task 1 SAF/Axes/XSDC2 <-> CX2020 (EtherCAT)/Term 1 (EK1200)/Term 2 (EK1122)/BOX-01 Coupler (EK1100)/BOX-03 ENC_X1_X2 (EL5042)
//     Enc/Inputs/In/nComState @bit 1 <-> WcState/InputToggle
//     Enc/Inputs/In/nComState <-> WcState/WcState
//     Enc/Inputs/In/nDataIn1 <-> FB Inputs Channel 2/Position
//     Enc/Inputs/In/nDcInputTime <-> InfoData/DcInputShift
//     Enc/Inputs/In/nState1 @bit 12 <-> FB Inputs Channel 2/Status/Diag
//     Enc/Inputs/In/nState1 @bit 1 <-> FB Inputs Channel 2/Status/Error
//     Enc/Inputs/In/nState1 @bit 14 <-> FB Inputs Channel 2/Status/Input cycle counter
//     Enc/Inputs/In/nState1 @bit 2 <-> FB Inputs Channel 2/Status/Ready
//     Enc/Inputs/In/nState1 @bit 13 <-> FB Inputs Channel 2/Status/TxPDO State
//     Enc/Inputs/In/nState1 <-> FB Inputs Channel 2/Status/Warning
//   NC-Task 1 SAF/Axes/XSDC2 <-> CX2020 (EtherCAT)/Term 1 (EK1200)/Term 2 (EK1122)/BOX-01 Coupler (EK1100)/BOX-10 DR_XSDC2 (EL7041-0052)
//     Drive/Inputs/In/nState1 @bit 3 <-> STM Status/Status/Error
//     Drive/Inputs/In/nState1 @bit 5 <-> STM Status/Status/Moving negative
//     Drive/Inputs/In/nState1 @bit 4 <-> STM Status/Status/Moving positive
//     Drive/Inputs/In/nState1 @bit 1 <-> STM Status/Status/Ready
//     Drive/Inputs/In/nState1 <-> STM Status/Status/Ready to enable
//     Drive/Inputs/In/nState1 @bit 6 <-> STM Status/Status/Torque reduced
//     Drive/Inputs/In/nState1 @bit 2 <-> STM Status/Status/Warning
//     Drive/Inputs/In/nState2 @bit 3 <-> STM Status/Status/Digital input 1
//     Drive/Inputs/In/nState2 @bit 4 <-> STM Status/Status/Digital input 2
//     Drive/Inputs/In/nState2 @bit 5 <-> STM Status/Status/Sync error
//     Drive/Inputs/In/nState2 @bit 7 <-> STM Status/Status/TxPDO Toggle
//     Drive/Inputs/In/nState4 @bit 1 <-> WcState/InputToggle
//     Drive/Inputs/In/nState4 <-> WcState/WcState
//     Drive/Outputs/Out/nCtrl1 <-> STM Control/Control/Enable
//     Drive/Outputs/Out/nCtrl1 @bit 2 <-> STM Control/Control/Reduce torque
//     Drive/Outputs/Out/nCtrl1 @bit 1 <-> STM Control/Control/Reset
//     Drive/Outputs/Out/nDataOut2[0] <-> STM Velocity/Velocity
//   NC-Task 1 SAF/Axes/YDF1 <-> CX2020 (EtherCAT)/Term 1 (EK1200)/Term 2 (EK1122)/Rack#2B-01 Coupler (EK1100)/Rack#2B-15 DR_YDF1 (EL7041-0052)
//     Drive/Inputs/In/nDcOutputTime <-> InfoData/DcOutputShift
//     Drive/Inputs/In/nState1 @bit 3 <-> STM Status/Status/Error
//     Drive/Inputs/In/nState1 @bit 5 <-> STM Status/Status/Moving negative
//     Drive/Inputs/In/nState1 @bit 4 <-> STM Status/Status/Moving positive
//     Drive/Inputs/In/nState1 @bit 1 <-> STM Status/Status/Ready
//     Drive/Inputs/In/nState1 <-> STM Status/Status/Ready to enable
//     Drive/Inputs/In/nState1 @bit 6 <-> STM Status/Status/Torque reduced
//     Drive/Inputs/In/nState1 @bit 2 <-> STM Status/Status/Warning
//     Drive/Inputs/In/nState2 @bit 3 <-> STM Status/Status/Digital input 1
//     Drive/Inputs/In/nState2 @bit 4 <-> STM Status/Status/Digital input 2
//     Drive/Inputs/In/nState2 @bit 5 <-> STM Status/Status/Sync error
//     Drive/Inputs/In/nState2 @bit 7 <-> STM Status/Status/TxPDO Toggle
//     Drive/Inputs/In/nState4 @bit 1 <-> WcState/InputToggle
//     Drive/Inputs/In/nState4 <-> WcState/WcState
//     Drive/Outputs/Out/nCtrl1 <-> STM Control/Control/Enable
//     Drive/Outputs/Out/nCtrl1 @bit 2 <-> STM Control/Control/Reduce torque
//     Drive/Outputs/Out/nCtrl1 @bit 1 <-> STM Control/Control/Reset
//     Drive/Outputs/Out/nDataOut2[0] <-> STM Velocity/Velocity
//   NC-Task 1 SAF/Axes/YDF2 <-> CX2020 (EtherCAT)/Term 1 (EK1200)/Term 2 (EK1122)/Rack#2B-01 Coupler (EK1100)/Rack#2B-16 DR_YDF2 (EL7041-0052)
//     Drive/Inputs/In/nState1 @bit 3 <-> STM Status/Status/Error
//     Drive/Inputs/In/nState1 @bit 5 <-> STM Status/Status/Moving negative
//     Drive/Inputs/In/nState1 @bit 4 <-> STM Status/Status/Moving positive
//     Drive/Inputs/In/nState1 @bit 1 <-> STM Status/Status/Ready
//     Drive/Inputs/In/nState1 <-> STM Status/Status/Ready to enable
//     Drive/Inputs/In/nState1 @bit 6 <-> STM Status/Status/Torque reduced
//     Drive/Inputs/In/nState1 @bit 2 <-> STM Status/Status/Warning
//     Drive/Inputs/In/nState2 @bit 3 <-> STM Status/Status/Digital input 1
//     Drive/Inputs/In/nState2 @bit 4 <-> STM Status/Status/Digital input 2
//     Drive/Inputs/In/nState2 @bit 5 <-> STM Status/Status/Sync error
//     Drive/Inputs/In/nState2 @bit 7 <-> STM Status/Status/TxPDO Toggle
//     Drive/Inputs/In/nState4 @bit 1 <-> WcState/InputToggle
//     Drive/Inputs/In/nState4 <-> WcState/WcState
//     Drive/Outputs/Out/nCtrl1 <-> STM Control/Control/Enable
//     Drive/Outputs/Out/nCtrl1 @bit 2 <-> STM Control/Control/Reduce torque
//     Drive/Outputs/Out/nCtrl1 @bit 1 <-> STM Control/Control/Reset
//     Drive/Outputs/Out/nDataOut2[0] <-> STM Velocity/Velocity
//   NC-Task 1 SAF/Axes/YDF3 <-> CX2020 (EtherCAT)/Term 1 (EK1200)/Term 2 (EK1122)/Rack#2B-01 Coupler (EK1100)/Rack#2B-19 DR_YDF3 (EL7041-0052)
//     Drive/Inputs/In/nState1 @bit 3 <-> STM Status/Status/Error
//     Drive/Inputs/In/nState1 @bit 5 <-> STM Status/Status/Moving negative
//     Drive/Inputs/In/nState1 @bit 4 <-> STM Status/Status/Moving positive
//     Drive/Inputs/In/nState1 @bit 1 <-> STM Status/Status/Ready
//     Drive/Inputs/In/nState1 <-> STM Status/Status/Ready to enable
//     Drive/Inputs/In/nState1 @bit 6 <-> STM Status/Status/Torque reduced
//     Drive/Inputs/In/nState1 @bit 2 <-> STM Status/Status/Warning
//     Drive/Inputs/In/nState2 @bit 3 <-> STM Status/Status/Digital input 1
//     Drive/Inputs/In/nState2 @bit 4 <-> STM Status/Status/Digital input 2
//     Drive/Inputs/In/nState2 @bit 5 <-> STM Status/Status/Sync error
//     Drive/Inputs/In/nState2 @bit 7 <-> STM Status/Status/TxPDO Toggle
//     Drive/Inputs/In/nState4 @bit 1 <-> WcState/InputToggle
//     Drive/Inputs/In/nState4 <-> WcState/WcState
//     Drive/Outputs/Out/nCtrl1 <-> STM Control/Control/Enable
//     Drive/Outputs/Out/nCtrl1 @bit 2 <-> STM Control/Control/Reduce torque
//     Drive/Outputs/Out/nCtrl1 @bit 1 <-> STM Control/Control/Reset
//     Drive/Outputs/Out/nDataOut2[0] <-> STM Velocity/Velocity
//   NC-Task 1 SAF/Axes/YF1 <-> CX2020 (EtherCAT)/Term 1 (EK1200)/Term 2 (EK1122)/BOX-01 Coupler (EK1100)/BOX-06 ENC_ZDC_YF1 (EL5042)
//     Enc/Inputs/In/nComState @bit 1 <-> WcState/InputToggle
//     Enc/Inputs/In/nComState <-> WcState/WcState
//     Enc/Inputs/In/nDataIn1 <-> FB Inputs Channel 2/Position
//     Enc/Inputs/In/nDcInputTime <-> InfoData/DcInputShift
//     Enc/Inputs/In/nState1 @bit 12 <-> FB Inputs Channel 2/Status/Diag
//     Enc/Inputs/In/nState1 @bit 1 <-> FB Inputs Channel 2/Status/Error
//     Enc/Inputs/In/nState1 @bit 14 <-> FB Inputs Channel 2/Status/Input cycle counter
//     Enc/Inputs/In/nState1 @bit 2 <-> FB Inputs Channel 2/Status/Ready
//     Enc/Inputs/In/nState1 @bit 13 <-> FB Inputs Channel 2/Status/TxPDO State
//     Enc/Inputs/In/nState1 <-> FB Inputs Channel 2/Status/Warning
//   NC-Task 1 SAF/Axes/YF1 <-> CX2020 (EtherCAT)/Term 1 (EK1200)/Term 2 (EK1122)/BOX-01 Coupler (EK1100)/BOX-20 DR_YF1 (EL7047)
//     Drive/Inputs/In/nState1 @bit 3 <-> STM Status/Status/Error
//     Drive/Inputs/In/nState1 @bit 7 <-> STM Status/Status/Motor stall
//     Drive/Inputs/In/nState1 @bit 5 <-> STM Status/Status/Moving negative
//     Drive/Inputs/In/nState1 @bit 4 <-> STM Status/Status/Moving positive
//     Drive/Inputs/In/nState1 @bit 1 <-> STM Status/Status/Ready
//     Drive/Inputs/In/nState1 <-> STM Status/Status/Ready to enable
//     Drive/Inputs/In/nState1 @bit 6 <-> STM Status/Status/Torque reduced
//     Drive/Inputs/In/nState1 @bit 2 <-> STM Status/Status/Warning
//     Drive/Inputs/In/nState2 @bit 3 <-> STM Status/Status/Digital input 1
//     Drive/Inputs/In/nState2 @bit 4 <-> STM Status/Status/Digital input 2
//     Drive/Inputs/In/nState2 @bit 5 <-> STM Status/Status/Sync error
//     Drive/Inputs/In/nState2 @bit 7 <-> STM Status/Status/TxPDO Toggle
//     Drive/Inputs/In/nState4 @bit 1 <-> WcState/InputToggle
//     Drive/Inputs/In/nState4 <-> WcState/WcState
//     Drive/Outputs/Out/nCtrl1 <-> STM Control/Control/Enable
//     Drive/Outputs/Out/nCtrl1 @bit 2 <-> STM Control/Control/Reduce torque
//     Drive/Outputs/Out/nCtrl1 @bit 1 <-> STM Control/Control/Reset
//     Drive/Outputs/Out/nCtrl2 @bit 3 <-> STM Control/Control/Digital output 1
//     Drive/Outputs/Out/nDataOut2[0] <-> STM Velocity/Velocity
//   NC-Task 1 SAF/Axes/YF2 <-> CX2020 (EtherCAT)/Term 1 (EK1200)/Term 2 (EK1122)/BOX-01 Coupler (EK1100)/BOX-07 ENC_YF2_ZF (EL5042)
//     Enc/Inputs/In/nComState @bit 1 <-> WcState/InputToggle
//     Enc/Inputs/In/nComState <-> WcState/WcState
//     Enc/Inputs/In/nDataIn1 <-> FB Inputs Channel 1/Position
//     Enc/Inputs/In/nDcInputTime <-> InfoData/DcInputShift
//     Enc/Inputs/In/nState1 @bit 12 <-> FB Inputs Channel 1/Status/Diag
//     Enc/Inputs/In/nState1 @bit 1 <-> FB Inputs Channel 1/Status/Error
//     Enc/Inputs/In/nState1 @bit 14 <-> FB Inputs Channel 1/Status/Input cycle counter
//     Enc/Inputs/In/nState1 @bit 2 <-> FB Inputs Channel 1/Status/Ready
//     Enc/Inputs/In/nState1 @bit 13 <-> FB Inputs Channel 1/Status/TxPDO State
//     Enc/Inputs/In/nState1 <-> FB Inputs Channel 1/Status/Warning
//   NC-Task 1 SAF/Axes/YF2 <-> CX2020 (EtherCAT)/Term 1 (EK1200)/Term 2 (EK1122)/BOX-01 Coupler (EK1100)/BOX-21 DR_YF2 (EL7047)
//     Drive/Inputs/In/nState1 @bit 3 <-> STM Status/Status/Error
//     Drive/Inputs/In/nState1 @bit 7 <-> STM Status/Status/Motor stall
//     Drive/Inputs/In/nState1 @bit 5 <-> STM Status/Status/Moving negative
//     Drive/Inputs/In/nState1 @bit 4 <-> STM Status/Status/Moving positive
//     Drive/Inputs/In/nState1 @bit 1 <-> STM Status/Status/Ready
//     Drive/Inputs/In/nState1 <-> STM Status/Status/Ready to enable
//     Drive/Inputs/In/nState1 @bit 6 <-> STM Status/Status/Torque reduced
//     Drive/Inputs/In/nState1 @bit 2 <-> STM Status/Status/Warning
//     Drive/Inputs/In/nState2 @bit 3 <-> STM Status/Status/Digital input 1
//     Drive/Inputs/In/nState2 @bit 4 <-> STM Status/Status/Digital input 2
//     Drive/Inputs/In/nState2 @bit 5 <-> STM Status/Status/Sync error
//     Drive/Inputs/In/nState2 @bit 7 <-> STM Status/Status/TxPDO Toggle
//     Drive/Inputs/In/nState4 @bit 1 <-> WcState/InputToggle
//     Drive/Inputs/In/nState4 <-> WcState/WcState
//     Drive/Outputs/Out/nCtrl1 <-> STM Control/Control/Enable
//     Drive/Outputs/Out/nCtrl1 @bit 2 <-> STM Control/Control/Reduce torque
//     Drive/Outputs/Out/nCtrl1 @bit 1 <-> STM Control/Control/Reset
//     Drive/Outputs/Out/nCtrl2 @bit 3 <-> STM Control/Control/Digital output 1
//     Drive/Outputs/Out/nDataOut2[0] <-> STM Velocity/Velocity
//   NC-Task 1 SAF/Axes/YG1 <-> CX2020 (EtherCAT)/Term 1 (EK1200)/Term 2 (EK1122)/Rack#2A-01 Coupler (EK1100)/Rack#2A-10 DR_YG1 (EL7041-0052)
//     Drive/Inputs/In/nDcOutputTime <-> InfoData/DcOutputShift
//     Drive/Inputs/In/nState1 @bit 3 <-> STM Status/Status/Error
//     Drive/Inputs/In/nState1 @bit 5 <-> STM Status/Status/Moving negative
//     Drive/Inputs/In/nState1 @bit 4 <-> STM Status/Status/Moving positive
//     Drive/Inputs/In/nState1 @bit 1 <-> STM Status/Status/Ready
//     Drive/Inputs/In/nState1 <-> STM Status/Status/Ready to enable
//     Drive/Inputs/In/nState1 @bit 6 <-> STM Status/Status/Torque reduced
//     Drive/Inputs/In/nState1 @bit 2 <-> STM Status/Status/Warning
//     Drive/Inputs/In/nState2 @bit 3 <-> STM Status/Status/Digital input 1
//     Drive/Inputs/In/nState2 @bit 4 <-> STM Status/Status/Digital input 2
//     Drive/Inputs/In/nState2 @bit 5 <-> STM Status/Status/Sync error
//     Drive/Inputs/In/nState2 @bit 7 <-> STM Status/Status/TxPDO Toggle
//     Drive/Inputs/In/nState4 @bit 1 <-> WcState/InputToggle
//     Drive/Inputs/In/nState4 <-> WcState/WcState
//     Drive/Outputs/Out/nCtrl1 <-> STM Control/Control/Enable
//     Drive/Outputs/Out/nCtrl1 @bit 2 <-> STM Control/Control/Reduce torque
//     Drive/Outputs/Out/nCtrl1 @bit 1 <-> STM Control/Control/Reset
//     Drive/Outputs/Out/nDataOut2[0] <-> STM Velocity/Velocity
//   NC-Task 1 SAF/Axes/YG1 <-> CX2020 (EtherCAT)/Term 1 (EK1200)/Term 2 (EK1122)/Rack#2B-01 Coupler (EK1100)/Rack#2B-10 ENC_YG1_YG2 (EL5042)
//     Enc/Inputs/In/nComState @bit 1 <-> WcState/InputToggle
//     Enc/Inputs/In/nComState <-> WcState/WcState
//     Enc/Inputs/In/nDataIn1 <-> FB Inputs Channel 1/Position
//     Enc/Inputs/In/nDcInputTime <-> InfoData/DcInputShift
//     Enc/Inputs/In/nState1 @bit 12 <-> FB Inputs Channel 1/Status/Diag
//     Enc/Inputs/In/nState1 @bit 1 <-> FB Inputs Channel 1/Status/Error
//     Enc/Inputs/In/nState1 @bit 14 <-> FB Inputs Channel 1/Status/Input cycle counter
//     Enc/Inputs/In/nState1 @bit 2 <-> FB Inputs Channel 1/Status/Ready
//     Enc/Inputs/In/nState1 @bit 13 <-> FB Inputs Channel 1/Status/TxPDO State
//     Enc/Inputs/In/nState1 <-> FB Inputs Channel 1/Status/Warning
//   NC-Task 1 SAF/Axes/YG2 <-> CX2020 (EtherCAT)/Term 1 (EK1200)/Term 2 (EK1122)/Rack#2A-01 Coupler (EK1100)/Rack#2A-11 DR_YG2 (EL7041-0052)
//     Drive/Inputs/In/nState1 @bit 3 <-> STM Status/Status/Error
//     Drive/Inputs/In/nState1 @bit 5 <-> STM Status/Status/Moving negative
//     Drive/Inputs/In/nState1 @bit 4 <-> STM Status/Status/Moving positive
//     Drive/Inputs/In/nState1 @bit 1 <-> STM Status/Status/Ready
//     Drive/Inputs/In/nState1 <-> STM Status/Status/Ready to enable
//     Drive/Inputs/In/nState1 @bit 6 <-> STM Status/Status/Torque reduced
//     Drive/Inputs/In/nState1 @bit 2 <-> STM Status/Status/Warning
//     Drive/Inputs/In/nState2 @bit 5 <-> STM Status/Status/Sync error
//     Drive/Inputs/In/nState2 @bit 7 <-> STM Status/Status/TxPDO Toggle
//     Drive/Inputs/In/nState4 @bit 1 <-> WcState/InputToggle
//     Drive/Inputs/In/nState4 <-> WcState/WcState
//     Drive/Outputs/Out/nCtrl1 <-> STM Control/Control/Enable
//     Drive/Outputs/Out/nCtrl1 @bit 2 <-> STM Control/Control/Reduce torque
//     Drive/Outputs/Out/nCtrl1 @bit 1 <-> STM Control/Control/Reset
//     Drive/Outputs/Out/nDataOut2[0] <-> STM Velocity/Velocity
//   NC-Task 1 SAF/Axes/YG2 <-> CX2020 (EtherCAT)/Term 1 (EK1200)/Term 2 (EK1122)/Rack#2B-01 Coupler (EK1100)/Rack#2B-10 ENC_YG1_YG2 (EL5042)
//     Enc/Inputs/In/nComState @bit 1 <-> WcState/InputToggle
//     Enc/Inputs/In/nComState <-> WcState/WcState
//     Enc/Inputs/In/nDataIn1 <-> FB Inputs Channel 2/Position
//     Enc/Inputs/In/nDcInputTime <-> InfoData/DcInputShift
//     Enc/Inputs/In/nState1 @bit 12 <-> FB Inputs Channel 2/Status/Diag
//     Enc/Inputs/In/nState1 @bit 1 <-> FB Inputs Channel 2/Status/Error
//     Enc/Inputs/In/nState1 @bit 14 <-> FB Inputs Channel 2/Status/Input cycle counter
//     Enc/Inputs/In/nState1 @bit 2 <-> FB Inputs Channel 2/Status/Ready
//     Enc/Inputs/In/nState1 @bit 13 <-> FB Inputs Channel 2/Status/TxPDO State
//     Enc/Inputs/In/nState1 <-> FB Inputs Channel 2/Status/Warning
//   NC-Task 1 SAF/Axes/YG3 <-> CX2020 (EtherCAT)/Term 1 (EK1200)/Term 2 (EK1122)/Rack#2A-01 Coupler (EK1100)/Rack#2A-12 DR_YG3 (EL7041-0052)
//     Drive/Inputs/In/nState1 @bit 3 <-> STM Status/Status/Error
//     Drive/Inputs/In/nState1 @bit 5 <-> STM Status/Status/Moving negative
//     Drive/Inputs/In/nState1 @bit 4 <-> STM Status/Status/Moving positive
//     Drive/Inputs/In/nState1 @bit 1 <-> STM Status/Status/Ready
//     Drive/Inputs/In/nState1 <-> STM Status/Status/Ready to enable
//     Drive/Inputs/In/nState1 @bit 6 <-> STM Status/Status/Torque reduced
//     Drive/Inputs/In/nState1 @bit 2 <-> STM Status/Status/Warning
//     Drive/Inputs/In/nState2 @bit 5 <-> STM Status/Status/Sync error
//     Drive/Inputs/In/nState2 @bit 7 <-> STM Status/Status/TxPDO Toggle
//     Drive/Inputs/In/nState4 @bit 1 <-> WcState/InputToggle
//     Drive/Inputs/In/nState4 <-> WcState/WcState
//     Drive/Outputs/Out/nCtrl1 <-> STM Control/Control/Enable
//     Drive/Outputs/Out/nCtrl1 @bit 2 <-> STM Control/Control/Reduce torque
//     Drive/Outputs/Out/nCtrl1 @bit 1 <-> STM Control/Control/Reset
//     Drive/Outputs/Out/nDataOut2[0] <-> STM Velocity/Velocity
//   NC-Task 1 SAF/Axes/YG3 <-> CX2020 (EtherCAT)/Term 1 (EK1200)/Term 2 (EK1122)/Rack#2B-01 Coupler (EK1100)/Rack#2B-11 ENC_YG3_X1PM (EL5042)
//     Enc/Inputs/In/nComState @bit 1 <-> WcState/InputToggle
//     Enc/Inputs/In/nComState <-> WcState/WcState
//     Enc/Inputs/In/nDataIn1 <-> FB Inputs Channel 1/Position
//     Enc/Inputs/In/nDcInputTime <-> InfoData/DcInputShift
//     Enc/Inputs/In/nState1 @bit 12 <-> FB Inputs Channel 1/Status/Diag
//     Enc/Inputs/In/nState1 @bit 1 <-> FB Inputs Channel 1/Status/Error
//     Enc/Inputs/In/nState1 @bit 14 <-> FB Inputs Channel 1/Status/Input cycle counter
//     Enc/Inputs/In/nState1 @bit 2 <-> FB Inputs Channel 1/Status/Ready
//     Enc/Inputs/In/nState1 @bit 13 <-> FB Inputs Channel 1/Status/TxPDO State
//     Enc/Inputs/In/nState1 <-> FB Inputs Channel 1/Status/Warning
//   NC-Task 1 SAF/Axes/YS1 <-> CX2020 (EtherCAT)/Term 1 (EK1200)/Term 2 (EK1122)/Rack#2A-01 Coupler (EK1100)/Rack#2A-05 DR_YS1 (EL7041-0052)
//     Drive/Inputs/In/nState1 @bit 3 <-> STM Status/Status/Error
//     Drive/Inputs/In/nState1 @bit 5 <-> STM Status/Status/Moving negative
//     Drive/Inputs/In/nState1 @bit 4 <-> STM Status/Status/Moving positive
//     Drive/Inputs/In/nState1 @bit 1 <-> STM Status/Status/Ready
//     Drive/Inputs/In/nState1 <-> STM Status/Status/Ready to enable
//     Drive/Inputs/In/nState1 @bit 6 <-> STM Status/Status/Torque reduced
//     Drive/Inputs/In/nState1 @bit 2 <-> STM Status/Status/Warning
//     Drive/Inputs/In/nState2 @bit 3 <-> STM Status/Status/Digital input 1
//     Drive/Inputs/In/nState2 @bit 4 <-> STM Status/Status/Digital input 2
//     Drive/Inputs/In/nState2 @bit 5 <-> STM Status/Status/Sync error
//     Drive/Inputs/In/nState2 @bit 7 <-> STM Status/Status/TxPDO Toggle
//     Drive/Inputs/In/nState4 @bit 1 <-> WcState/InputToggle
//     Drive/Inputs/In/nState4 <-> WcState/WcState
//     Drive/Outputs/Out/nCtrl1 <-> STM Control/Control/Enable
//     Drive/Outputs/Out/nCtrl1 @bit 2 <-> STM Control/Control/Reduce torque
//     Drive/Outputs/Out/nCtrl1 @bit 1 <-> STM Control/Control/Reset
//     Drive/Outputs/Out/nDataOut2[0] <-> STM Velocity/Velocity
//   NC-Task 1 SAF/Axes/YS1 <-> CX2020 (EtherCAT)/Term 1 (EK1200)/Term 2 (EK1122)/Rack#2B-01 Coupler (EK1100)/Rack#2B-08 ENC_Y1_Y2 (EL5042)
//     Enc/Inputs/In/nComState @bit 1 <-> WcState/InputToggle
//     Enc/Inputs/In/nComState <-> WcState/WcState
//     Enc/Inputs/In/nDataIn1 <-> FB Inputs Channel 1/Position
//     Enc/Inputs/In/nDcInputTime <-> InfoData/DcInputShift
//     Enc/Inputs/In/nState1 @bit 12 <-> FB Inputs Channel 1/Status/Diag
//     Enc/Inputs/In/nState1 @bit 1 <-> FB Inputs Channel 1/Status/Error
//     Enc/Inputs/In/nState1 @bit 14 <-> FB Inputs Channel 1/Status/Input cycle counter
//     Enc/Inputs/In/nState1 @bit 2 <-> FB Inputs Channel 1/Status/Ready
//     Enc/Inputs/In/nState1 @bit 13 <-> FB Inputs Channel 1/Status/TxPDO State
//     Enc/Inputs/In/nState1 <-> FB Inputs Channel 1/Status/Warning
//   NC-Task 1 SAF/Axes/YS2 <-> CX2020 (EtherCAT)/Term 1 (EK1200)/Term 2 (EK1122)/Rack#2A-01 Coupler (EK1100)/Rack#2A-06 DR_YS2 (EL7041-0052)
//     Drive/Inputs/In/nState1 @bit 3 <-> STM Status/Status/Error
//     Drive/Inputs/In/nState1 @bit 5 <-> STM Status/Status/Moving negative
//     Drive/Inputs/In/nState1 @bit 4 <-> STM Status/Status/Moving positive
//     Drive/Inputs/In/nState1 @bit 1 <-> STM Status/Status/Ready
//     Drive/Inputs/In/nState1 <-> STM Status/Status/Ready to enable
//     Drive/Inputs/In/nState1 @bit 6 <-> STM Status/Status/Torque reduced
//     Drive/Inputs/In/nState1 @bit 2 <-> STM Status/Status/Warning
//     Drive/Inputs/In/nState2 @bit 3 <-> STM Status/Status/Digital input 1
//     Drive/Inputs/In/nState2 @bit 4 <-> STM Status/Status/Digital input 2
//     Drive/Inputs/In/nState2 @bit 5 <-> STM Status/Status/Sync error
//     Drive/Inputs/In/nState2 @bit 7 <-> STM Status/Status/TxPDO Toggle
//     Drive/Inputs/In/nState4 @bit 1 <-> WcState/InputToggle
//     Drive/Inputs/In/nState4 <-> WcState/WcState
//     Drive/Outputs/Out/nCtrl1 <-> STM Control/Control/Enable
//     Drive/Outputs/Out/nCtrl1 @bit 2 <-> STM Control/Control/Reduce torque
//     Drive/Outputs/Out/nCtrl1 @bit 1 <-> STM Control/Control/Reset
//     Drive/Outputs/Out/nDataOut2[0] <-> STM Velocity/Velocity
//   NC-Task 1 SAF/Axes/YS2 <-> CX2020 (EtherCAT)/Term 1 (EK1200)/Term 2 (EK1122)/Rack#2B-01 Coupler (EK1100)/Rack#2B-08 ENC_Y1_Y2 (EL5042)
//     Enc/Inputs/In/nComState @bit 1 <-> WcState/InputToggle
//     Enc/Inputs/In/nComState <-> WcState/WcState
//     Enc/Inputs/In/nDataIn1 <-> FB Inputs Channel 2/Position
//     Enc/Inputs/In/nDcInputTime <-> InfoData/DcInputShift
//     Enc/Inputs/In/nState1 @bit 12 <-> FB Inputs Channel 2/Status/Diag
//     Enc/Inputs/In/nState1 @bit 1 <-> FB Inputs Channel 2/Status/Error
//     Enc/Inputs/In/nState1 @bit 14 <-> FB Inputs Channel 2/Status/Input cycle counter
//     Enc/Inputs/In/nState1 @bit 2 <-> FB Inputs Channel 2/Status/Ready
//     Enc/Inputs/In/nState1 @bit 13 <-> FB Inputs Channel 2/Status/TxPDO State
//     Enc/Inputs/In/nState1 <-> FB Inputs Channel 2/Status/Warning
//   NC-Task 1 SAF/Axes/YSDC1 <-> CX2020 (EtherCAT)/Term 1 (EK1200)/Term 2 (EK1122)/BOX-01 Coupler (EK1100)/BOX-04 ENC_Y1_Y2 (EL5042)
//     Enc/Inputs/In/nComState @bit 1 <-> WcState/InputToggle
//     Enc/Inputs/In/nComState <-> WcState/WcState
//     Enc/Inputs/In/nDataIn1 <-> FB Inputs Channel 1/Position
//     Enc/Inputs/In/nDcInputTime <-> InfoData/DcInputShift
//     Enc/Inputs/In/nState1 @bit 12 <-> FB Inputs Channel 1/Status/Diag
//     Enc/Inputs/In/nState1 @bit 1 <-> FB Inputs Channel 1/Status/Error
//     Enc/Inputs/In/nState1 @bit 14 <-> FB Inputs Channel 1/Status/Input cycle counter
//     Enc/Inputs/In/nState1 @bit 2 <-> FB Inputs Channel 1/Status/Ready
//     Enc/Inputs/In/nState1 @bit 13 <-> FB Inputs Channel 1/Status/TxPDO State
//     Enc/Inputs/In/nState1 <-> FB Inputs Channel 1/Status/Warning
//   NC-Task 1 SAF/Axes/YSDC1 <-> CX2020 (EtherCAT)/Term 1 (EK1200)/Term 2 (EK1122)/BOX-01 Coupler (EK1100)/BOX-11 DR_YSDC1 (EL7041-0052)
//     Drive/Inputs/In/nState1 @bit 3 <-> STM Status/Status/Error
//     Drive/Inputs/In/nState1 @bit 5 <-> STM Status/Status/Moving negative
//     Drive/Inputs/In/nState1 @bit 4 <-> STM Status/Status/Moving positive
//     Drive/Inputs/In/nState1 @bit 1 <-> STM Status/Status/Ready
//     Drive/Inputs/In/nState1 <-> STM Status/Status/Ready to enable
//     Drive/Inputs/In/nState1 @bit 6 <-> STM Status/Status/Torque reduced
//     Drive/Inputs/In/nState1 @bit 2 <-> STM Status/Status/Warning
//     Drive/Inputs/In/nState2 @bit 3 <-> STM Status/Status/Digital input 1
//     Drive/Inputs/In/nState2 @bit 4 <-> STM Status/Status/Digital input 2
//     Drive/Inputs/In/nState2 @bit 5 <-> STM Status/Status/Sync error
//     Drive/Inputs/In/nState2 @bit 7 <-> STM Status/Status/TxPDO Toggle
//     Drive/Inputs/In/nState4 @bit 1 <-> WcState/InputToggle
//     Drive/Inputs/In/nState4 <-> WcState/WcState
//     Drive/Outputs/Out/nCtrl1 <-> STM Control/Control/Enable
//     Drive/Outputs/Out/nCtrl1 @bit 2 <-> STM Control/Control/Reduce torque
//     Drive/Outputs/Out/nCtrl1 @bit 1 <-> STM Control/Control/Reset
//     Drive/Outputs/Out/nDataOut2[0] <-> STM Velocity/Velocity
//   NC-Task 1 SAF/Axes/YSDC2 <-> CX2020 (EtherCAT)/Term 1 (EK1200)/Term 2 (EK1122)/BOX-01 Coupler (EK1100)/BOX-04 ENC_Y1_Y2 (EL5042)
//     Enc/Inputs/In/nComState @bit 1 <-> WcState/InputToggle
//     Enc/Inputs/In/nComState <-> WcState/WcState
//     Enc/Inputs/In/nDataIn1 <-> FB Inputs Channel 2/Position
//     Enc/Inputs/In/nDcInputTime <-> InfoData/DcInputShift
//     Enc/Inputs/In/nState1 @bit 12 <-> FB Inputs Channel 2/Status/Diag
//     Enc/Inputs/In/nState1 @bit 1 <-> FB Inputs Channel 2/Status/Error
//     Enc/Inputs/In/nState1 @bit 14 <-> FB Inputs Channel 2/Status/Input cycle counter
//     Enc/Inputs/In/nState1 @bit 2 <-> FB Inputs Channel 2/Status/Ready
//     Enc/Inputs/In/nState1 @bit 13 <-> FB Inputs Channel 2/Status/TxPDO State
//     Enc/Inputs/In/nState1 <-> FB Inputs Channel 2/Status/Warning
//   NC-Task 1 SAF/Axes/YSDC2 <-> CX2020 (EtherCAT)/Term 1 (EK1200)/Term 2 (EK1122)/BOX-01 Coupler (EK1100)/BOX-12 DR_YSDC2 (EL7041-0052)
//     Drive/Inputs/In/nState1 @bit 3 <-> STM Status/Status/Error
//     Drive/Inputs/In/nState1 @bit 5 <-> STM Status/Status/Moving negative
//     Drive/Inputs/In/nState1 @bit 4 <-> STM Status/Status/Moving positive
//     Drive/Inputs/In/nState1 @bit 1 <-> STM Status/Status/Ready
//     Drive/Inputs/In/nState1 <-> STM Status/Status/Ready to enable
//     Drive/Inputs/In/nState1 @bit 6 <-> STM Status/Status/Torque reduced
//     Drive/Inputs/In/nState1 @bit 2 <-> STM Status/Status/Warning
//     Drive/Inputs/In/nState2 @bit 3 <-> STM Status/Status/Digital input 1
//     Drive/Inputs/In/nState2 @bit 4 <-> STM Status/Status/Digital input 2
//     Drive/Inputs/In/nState2 @bit 5 <-> STM Status/Status/Sync error
//     Drive/Inputs/In/nState2 @bit 7 <-> STM Status/Status/TxPDO Toggle
//     Drive/Inputs/In/nState4 @bit 1 <-> WcState/InputToggle
//     Drive/Inputs/In/nState4 <-> WcState/WcState
//     Drive/Outputs/Out/nCtrl1 <-> STM Control/Control/Enable
//     Drive/Outputs/Out/nCtrl1 @bit 2 <-> STM Control/Control/Reduce torque
//     Drive/Outputs/Out/nCtrl1 @bit 1 <-> STM Control/Control/Reset
//     Drive/Outputs/Out/nDataOut2[0] <-> STM Velocity/Velocity
//   NC-Task 1 SAF/Axes/ZDC <-> CX2020 (EtherCAT)/Term 1 (EK1200)/Term 2 (EK1122)/BOX-01 Coupler (EK1100)/BOX-06 ENC_ZDC_YF1 (EL5042)
//     Enc/Inputs/In/nComState @bit 1 <-> WcState/InputToggle
//     Enc/Inputs/In/nComState <-> WcState/WcState
//     Enc/Inputs/In/nDataIn1 <-> FB Inputs Channel 1/Position
//     Enc/Inputs/In/nState1 @bit 12 <-> FB Inputs Channel 1/Status/Diag
//     Enc/Inputs/In/nState1 @bit 1 <-> FB Inputs Channel 1/Status/Error
//     Enc/Inputs/In/nState1 @bit 14 <-> FB Inputs Channel 1/Status/Input cycle counter
//     Enc/Inputs/In/nState1 @bit 2 <-> FB Inputs Channel 1/Status/Ready
//     Enc/Inputs/In/nState1 @bit 13 <-> FB Inputs Channel 1/Status/TxPDO State
//     Enc/Inputs/In/nState1 <-> FB Inputs Channel 1/Status/Warning
//   NC-Task 1 SAF/Axes/ZDC <-> CX2020 (EtherCAT)/Term 1 (EK1200)/Term 2 (EK1122)/BOX-01 Coupler (EK1100)/BOX-16 DR_ZDC (EL7041-0052)
//     Drive/Inputs/In/nState1 @bit 3 <-> STM Status/Status/Error
//     Drive/Inputs/In/nState1 @bit 5 <-> STM Status/Status/Moving negative
//     Drive/Inputs/In/nState1 @bit 4 <-> STM Status/Status/Moving positive
//     Drive/Inputs/In/nState1 @bit 1 <-> STM Status/Status/Ready
//     Drive/Inputs/In/nState1 <-> STM Status/Status/Ready to enable
//     Drive/Inputs/In/nState1 @bit 6 <-> STM Status/Status/Torque reduced
//     Drive/Inputs/In/nState1 @bit 2 <-> STM Status/Status/Warning
//     Drive/Inputs/In/nState2 @bit 3 <-> STM Status/Status/Digital input 1
//     Drive/Inputs/In/nState2 @bit 4 <-> STM Status/Status/Digital input 2
//     Drive/Inputs/In/nState2 @bit 5 <-> STM Status/Status/Sync error
//     Drive/Inputs/In/nState2 @bit 7 <-> STM Status/Status/TxPDO Toggle
//     Drive/Inputs/In/nState4 @bit 1 <-> WcState/InputToggle
//     Drive/Inputs/In/nState4 <-> WcState/WcState
//     Drive/Outputs/Out/nCtrl1 <-> STM Control/Control/Enable
//     Drive/Outputs/Out/nCtrl1 @bit 2 <-> STM Control/Control/Reduce torque
//     Drive/Outputs/Out/nCtrl1 @bit 1 <-> STM Control/Control/Reset
//     Drive/Outputs/Out/nDataOut2[0] <-> STM Velocity/Velocity
//   NC-Task 1 SAF/Axes/ZF <-> CX2020 (EtherCAT)/Term 1 (EK1200)/Term 2 (EK1122)/BOX-01 Coupler (EK1100)/BOX-07 ENC_YF2_ZF (EL5042)
//     Enc/Inputs/In/nComState @bit 1 <-> WcState/InputToggle
//     Enc/Inputs/In/nComState <-> WcState/WcState
//     Enc/Inputs/In/nDataIn1 <-> FB Inputs Channel 2/Position
//     Enc/Inputs/In/nDcInputTime <-> InfoData/DcInputShift
//     Enc/Inputs/In/nState1 @bit 12 <-> FB Inputs Channel 2/Status/Diag
//     Enc/Inputs/In/nState1 @bit 1 <-> FB Inputs Channel 2/Status/Error
//     Enc/Inputs/In/nState1 @bit 14 <-> FB Inputs Channel 2/Status/Input cycle counter
//     Enc/Inputs/In/nState1 @bit 2 <-> FB Inputs Channel 2/Status/Ready
//     Enc/Inputs/In/nState1 @bit 13 <-> FB Inputs Channel 2/Status/TxPDO State
//     Enc/Inputs/In/nState1 <-> FB Inputs Channel 2/Status/Warning
//   NC-Task 1 SAF/Axes/ZF <-> CX2020 (EtherCAT)/Term 1 (EK1200)/Term 2 (EK1122)/Rack#2B-01 Coupler (EK1100)/Rack#2B-20 DR_ZF (EL7047)
//     Drive/Inputs/In/nState1 @bit 3 <-> STM Status/Status/Error
//     Drive/Inputs/In/nState1 @bit 7 <-> STM Status/Status/Motor stall
//     Drive/Inputs/In/nState1 @bit 5 <-> STM Status/Status/Moving negative
//     Drive/Inputs/In/nState1 @bit 4 <-> STM Status/Status/Moving positive
//     Drive/Inputs/In/nState1 @bit 1 <-> STM Status/Status/Ready
//     Drive/Inputs/In/nState1 <-> STM Status/Status/Ready to enable
//     Drive/Inputs/In/nState1 @bit 6 <-> STM Status/Status/Torque reduced
//     Drive/Inputs/In/nState1 @bit 2 <-> STM Status/Status/Warning
//     Drive/Inputs/In/nState2 @bit 3 <-> STM Status/Status/Digital input 1
//     Drive/Inputs/In/nState2 @bit 4 <-> STM Status/Status/Digital input 2
//     Drive/Inputs/In/nState2 @bit 5 <-> STM Status/Status/Sync error
//     Drive/Inputs/In/nState2 @bit 7 <-> STM Status/Status/TxPDO Toggle
//     Drive/Inputs/In/nState4 @bit 1 <-> WcState/InputToggle
//     Drive/Inputs/In/nState4 <-> WcState/WcState
//     Drive/Outputs/Out/nCtrl1 <-> STM Control/Control/Enable
//     Drive/Outputs/Out/nCtrl1 @bit 2 <-> STM Control/Control/Reduce torque
//     Drive/Outputs/Out/nCtrl1 @bit 1 <-> STM Control/Control/Reset
//     Drive/Outputs/Out/nCtrl2 @bit 3 <-> STM Control/Control/Digital output 1
//     Drive/Outputs/Out/nDataOut2[0] <-> STM Velocity/Velocity
//   Motion/Motion Instance <-> CX2020 (EtherCAT)/Term 1 (EK1200)/Term 2 (EK1122)/BOX-01 Coupler (EK1100)/BOX-03 ENC_X1_X2 (EL5042)
//     PlcTask Inputs/GVL_Main.M18.nRawEncoderULINT <-> FB Inputs Channel 1/Position
//     PlcTask Inputs/GVL_Main.M19.nRawEncoderULINT <-> FB Inputs Channel 2/Position
//   Motion/Motion Instance <-> CX2020 (EtherCAT)/Term 1 (EK1200)/Term 2 (EK1122)/BOX-01 Coupler (EK1100)/BOX-04 ENC_Y1_Y2 (EL5042)
//     PlcTask Inputs/GVL_Main.M20.nRawEncoderULINT <-> FB Inputs Channel 1/Position
//     PlcTask Inputs/GVL_Main.M21.nRawEncoderULINT <-> FB Inputs Channel 1/Position
//   Motion/Motion Instance <-> CX2020 (EtherCAT)/Term 1 (EK1200)/Term 2 (EK1122)/BOX-01 Coupler (EK1100)/BOX-05 ENC_XDC_RyDC (EL5042)
//     PlcTask Inputs/GVL_Main.M22.nRawEncoderULINT <-> FB Inputs Channel 1/Position
//     PlcTask Inputs/GVL_Main.M23.nRawEncoderULINT <-> FB Inputs Channel 2/Position
//   Motion/Motion Instance <-> CX2020 (EtherCAT)/Term 1 (EK1200)/Term 2 (EK1122)/BOX-01 Coupler (EK1100)/BOX-06 ENC_ZDC_YF1 (EL5042)
//     PlcTask Inputs/GVL_Main.M24.nRawEncoderULINT <-> FB Inputs Channel 1/Position
//     PlcTask Inputs/GVL_Main.M25.nRawEncoderULINT <-> FB Inputs Channel 2/Position
//     PlcTask Inputs/PRG_DET_ARM.stRenishawAbsEncMaster.Count <-> FB Inputs Channel 2/Position
//   Motion/Motion Instance <-> CX2020 (EtherCAT)/Term 1 (EK1200)/Term 2 (EK1122)/BOX-01 Coupler (EK1100)/BOX-07 ENC_YF2_ZF (EL5042)
//     PlcTask Inputs/GVL_Main.M26.nRawEncoderULINT <-> FB Inputs Channel 1/Position
//     PlcTask Inputs/GVL_Main.M27.nRawEncoderULINT <-> FB Inputs Channel 2/Position
//     PlcTask Inputs/PRG_DET_ARM.stRenishawAbsEncSlave.Count <-> FB Inputs Channel 1/Position
//   Motion/Motion Instance <-> CX2020 (EtherCAT)/Term 1 (EK1200)/Term 2 (EK1122)/BOX-01 Coupler (EK1100)/BOX-09 DR_XSDC1 (EL7041-0052)
//     PlcTask Inputs/GVL_Main.M18.bLimitBackwardEnable <-> STM Status/Status/Digital input 2
//     PlcTask Inputs/GVL_Main.M18.bLimitForwardEnable <-> STM Status/Status/Digital input 1
//   Motion/Motion Instance <-> CX2020 (EtherCAT)/Term 1 (EK1200)/Term 2 (EK1122)/BOX-01 Coupler (EK1100)/BOX-10 DR_XSDC2 (EL7041-0052)
//     PlcTask Inputs/GVL_Main.M19.bLimitBackwardEnable <-> STM Status/Status/Digital input 2
//     PlcTask Inputs/GVL_Main.M19.bLimitForwardEnable <-> STM Status/Status/Digital input 1
//   Motion/Motion Instance <-> CX2020 (EtherCAT)/Term 1 (EK1200)/Term 2 (EK1122)/BOX-01 Coupler (EK1100)/BOX-11 DR_YSDC1 (EL7041-0052)
//     PlcTask Inputs/GVL_Main.M20.bLimitBackwardEnable <-> STM Status/Status/Digital input 2
//     PlcTask Inputs/GVL_Main.M20.bLimitForwardEnable <-> STM Status/Status/Digital input 1
//   Motion/Motion Instance <-> CX2020 (EtherCAT)/Term 1 (EK1200)/Term 2 (EK1122)/BOX-01 Coupler (EK1100)/BOX-12 DR_YSDC2 (EL7041-0052)
//     PlcTask Inputs/GVL_Main.M21.bLimitBackwardEnable <-> STM Status/Status/Digital input 2
//     PlcTask Inputs/GVL_Main.M21.bLimitForwardEnable <-> STM Status/Status/Digital input 1
//   Motion/Motion Instance <-> CX2020 (EtherCAT)/Term 1 (EK1200)/Term 2 (EK1122)/BOX-01 Coupler (EK1100)/BOX-14 DR_XDC (EL7041-0052)
//     PlcTask Inputs/GVL_Main.M22.bLimitBackwardEnable <-> STM Status/Status/Digital input 2
//     PlcTask Inputs/GVL_Main.M22.bLimitForwardEnable <-> STM Status/Status/Digital input 1
//   Motion/Motion Instance <-> CX2020 (EtherCAT)/Term 1 (EK1200)/Term 2 (EK1122)/BOX-01 Coupler (EK1100)/BOX-15 DR_RyDC (EL7041-0052)
//     PlcTask Inputs/GVL_Main.M23.bLimitBackwardEnable <-> STM Status/Status/Digital input 2
//     PlcTask Inputs/GVL_Main.M23.bLimitForwardEnable <-> STM Status/Status/Digital input 1
//   Motion/Motion Instance <-> CX2020 (EtherCAT)/Term 1 (EK1200)/Term 2 (EK1122)/BOX-01 Coupler (EK1100)/BOX-16 DR_ZDC (EL7041-0052)
//     PlcTask Inputs/GVL_Main.M24.bLimitBackwardEnable <-> STM Status/Status/Digital input 2
//     PlcTask Inputs/GVL_Main.M24.bLimitForwardEnable <-> STM Status/Status/Digital input 1
//   Motion/Motion Instance <-> CX2020 (EtherCAT)/Term 1 (EK1200)/Term 2 (EK1122)/BOX-01 Coupler (EK1100)/BOX-19 MB_YF1_YF2 (EL2602)
//     PlcTask Outputs/GVL_Main.M25.bBrakeRelease <-> Channel 1/Output
//     PlcTask Outputs/GVL_Main.M26.bBrakeRelease <-> Channel 2/Output
//   Motion/Motion Instance <-> CX2020 (EtherCAT)/Term 1 (EK1200)/Term 2 (EK1122)/Rack#1A-01 Coupler (EK1100)/Rack#1A-02 SFIN (EL1918)
//     PlcTask Inputs/GVL_Main.M25.bLimitBackwardEnable <-> StandardInputs/Standard Out Var 11
//     PlcTask Inputs/GVL_Main.M26.bLimitBackwardEnable <-> StandardInputs/Standard Out Var 13
//     PlcTask Inputs/GVL_Main.M27.bLimitBackwardEnable <-> StandardInputs/Standard Out Var 15
//     PlcTask Inputs/GVL_Main.M25.bLimitForwardEnable <-> StandardInputs/Standard Out Var 10
//     PlcTask Inputs/GVL_Main.M26.bLimitForwardEnable <-> StandardInputs/Standard Out Var 12
//     PlcTask Inputs/GVL_Main.M27.bLimitForwardEnable <-> StandardInputs/Standard Out Var 14
//     PlcTask Inputs/GVL_Main.bESTOP <-> StandardInputs/Standard Out Var 18
//     PlcTask Outputs/PRG1_MAIN_PlcTask.bEnaIclk <-> StandardOutputs/Standard In Var 2
//     PlcTask Outputs/PRG1_MAIN_PlcTask.bEnaIclkErrAck <-> StandardOutputs/Standard In Var 1
//     PlcTask Outputs/PRG1_MAIN_PlcTask.bEnaIclkRestartESTOP <-> StandardOutputs/Standard In Var 9
//   Motion/Motion Instance <-> CX2020 (EtherCAT)/Term 1 (EK1200)/Term 2 (EK1122)/Rack#1A-01 Coupler (EK1100)/Rack#1A-04 DR_2Th (EL7047)
//     PlcTask Inputs/GVL_Main.M2.bLimitBackwardEnable <-> STM Status/Status/Digital input 2
//     PlcTask Inputs/GVL_Main.M2.bLimitForwardEnable <-> STM Status/Status/Digital input 1
//   Motion/Motion Instance <-> CX2020 (EtherCAT)/Term 1 (EK1200)/Term 2 (EK1122)/Rack#1A-01 Coupler (EK1100)/Rack#1A-05 MB_2Th (EL2602)
//     PlcTask Outputs/GVL_Main.M2.bBrakeRelease <-> Channel 1/Output
//   Motion/Motion Instance <-> CX2020 (EtherCAT)/Term 1 (EK1200)/Term 2 (EK1122)/Rack#1A-01 Coupler (EK1100)/Rack#1A-06 ENC_2Th (EL5042)
//     PlcTask Inputs/GVL_Main.M2.nRawEncoderULINT <-> FB Inputs Channel 1/Position
//   Motion/Motion Instance <-> CX2020 (EtherCAT)/Term 1 (EK1200)/Term 2 (EK1122)/Rack#1C_ServoDR (NCR-HD Series)
//     PlcTask Outputs/GVL_Main.iServoTorqueLimitNegative <-> 260th receive PDO Mapping/Negative torque limit value
//     PlcTask Outputs/GVL_Main.iServoTorqueLimitPositive <-> 260th receive PDO Mapping/Positive torque limit value
//   Motion/Motion Instance <-> CX2020 (EtherCAT)/Term 1 (EK1200)/Term 2 (EK1122)/Rack#2A-01 Coupler (EK1100)/Rack#2A-03 DR_XS1 (EL7041-0052)
//     PlcTask Inputs/GVL_Main.M3.bLimitBackwardEnable <-> STM Status/Status/Digital input 2
//     PlcTask Inputs/GVL_Main.M3.bLimitForwardEnable <-> STM Status/Status/Digital input 1
//   Motion/Motion Instance <-> CX2020 (EtherCAT)/Term 1 (EK1200)/Term 2 (EK1122)/Rack#2A-01 Coupler (EK1100)/Rack#2A-04 DR_XS2 (EL7041-0052)
//     PlcTask Inputs/GVL_Main.M4.bLimitBackwardEnable <-> STM Status/Status/Digital input 2
//     PlcTask Inputs/GVL_Main.M4.bLimitForwardEnable <-> STM Status/Status/Digital input 1
//   Motion/Motion Instance <-> CX2020 (EtherCAT)/Term 1 (EK1200)/Term 2 (EK1122)/Rack#2A-01 Coupler (EK1100)/Rack#2A-05 DR_YS1 (EL7041-0052)
//     PlcTask Inputs/GVL_Main.M5.bLimitBackwardEnable <-> STM Status/Status/Digital input 2
//     PlcTask Inputs/GVL_Main.M5.bLimitForwardEnable <-> STM Status/Status/Digital input 1
//   Motion/Motion Instance <-> CX2020 (EtherCAT)/Term 1 (EK1200)/Term 2 (EK1122)/Rack#2A-01 Coupler (EK1100)/Rack#2A-06 DR_YS2 (EL7041-0052)
//     PlcTask Inputs/GVL_Main.M6.bLimitBackwardEnable <-> STM Status/Status/Digital input 2
//     PlcTask Inputs/GVL_Main.M6.bLimitForwardEnable <-> STM Status/Status/Digital input 1
//   Motion/Motion Instance <-> CX2020 (EtherCAT)/Term 1 (EK1200)/Term 2 (EK1122)/Rack#2A-01 Coupler (EK1100)/Rack#2A-08 DR_RxG (EL7041-0052)
//     PlcTask Inputs/GVL_Main.M10.bLimitBackwardEnable <-> STM Status/Status/Digital input 2
//     PlcTask Inputs/GVL_Main.M10.bLimitForwardEnable <-> STM Status/Status/Digital input 1
//   Motion/Motion Instance <-> CX2020 (EtherCAT)/Term 1 (EK1200)/Term 2 (EK1122)/Rack#2A-01 Coupler (EK1100)/Rack#2A-09 DR_XG (EL7041-0052)
//     PlcTask Inputs/GVL_Main.M11.bLimitBackwardEnable <-> STM Status/Status/Digital input 2
//     PlcTask Inputs/GVL_Main.M11.bLimitForwardEnable <-> STM Status/Status/Digital input 1
//   Motion/Motion Instance <-> CX2020 (EtherCAT)/Term 1 (EK1200)/Term 2 (EK1122)/Rack#2A-01 Coupler (EK1100)/Rack#2A-10 DR_YG1 (EL7041-0052)
//     PlcTask Inputs/GVL_Main.M7.bLimitBackwardEnable <-> STM Status/Status/Digital input 2
//     PlcTask Inputs/GVL_Main.M7.bLimitForwardEnable <-> STM Status/Status/Digital input 1
//   Motion/Motion Instance <-> CX2020 (EtherCAT)/Term 1 (EK1200)/Term 2 (EK1122)/Rack#2A-01 Coupler (EK1100)/Rack#2A-11 DR_YG2 (EL7041-0052)
//     PlcTask Inputs/GVL_Main.M8.bLimitBackwardEnable <-> STM Status/Status/Digital input 2
//     PlcTask Inputs/GVL_Main.M8.bLimitForwardEnable <-> STM Status/Status/Digital input 1
//   Motion/Motion Instance <-> CX2020 (EtherCAT)/Term 1 (EK1200)/Term 2 (EK1122)/Rack#2A-01 Coupler (EK1100)/Rack#2A-12 DR_YG3 (EL7041-0052)
//     PlcTask Inputs/GVL_Main.M9.bLimitBackwardEnable <-> STM Status/Status/Digital input 2
//     PlcTask Inputs/GVL_Main.M9.bLimitForwardEnable <-> STM Status/Status/Digital input 1
//   Motion/Motion Instance <-> CX2020 (EtherCAT)/Term 1 (EK1200)/Term 2 (EK1122)/Rack#2A-01 Coupler (EK1100)/Rack#2A-14 DR_XPM1 (EL7041-0052)
//     PlcTask Inputs/GVL_Main.M12.bLimitBackwardEnable <-> STM Status/Status/Digital input 2
//     PlcTask Inputs/GVL_Main.M12.bLimitForwardEnable <-> STM Status/Status/Digital input 1
//   Motion/Motion Instance <-> CX2020 (EtherCAT)/Term 1 (EK1200)/Term 2 (EK1122)/Rack#2A-01 Coupler (EK1100)/Rack#2A-15 DR_XPM2 (EL7041-0052)
//     PlcTask Inputs/GVL_Main.M13.bLimitBackwardEnable <-> STM Status/Status/Digital input 2
//     PlcTask Inputs/GVL_Main.M13.bLimitForwardEnable <-> STM Status/Status/Digital input 1
//   Motion/Motion Instance <-> CX2020 (EtherCAT)/Term 1 (EK1200)/Term 2 (EK1122)/Rack#2A-01 Coupler (EK1100)/Rack#2A-16 DR_RzPM (EL7041-0052)
//     PlcTask Inputs/GVL_Main.M14.bLimitBackwardEnable <-> STM Status/Status/Digital input 2
//     PlcTask Inputs/GVL_Main.M14.bLimitForwardEnable <-> STM Status/Status/Digital input 1
//   Motion/Motion Instance <-> CX2020 (EtherCAT)/Term 1 (EK1200)/Term 2 (EK1122)/Rack#2B-01 Coupler (EK1100)/Rack#2B-03 AI_TiltSensor (EL3174-0002)
//     PlcTask Inputs/GVL_Sensor.stFrameP.iRawCnts <-> AI Standard Channel 4/Value
//     PlcTask Inputs/GVL_Sensor.stFrameR.iRawCnts <-> AI Standard Channel 3/Value
//     PlcTask Inputs/GVL_Sensor.stGraniteP.iRawCnts <-> AI Standard Channel 2/Value
//     PlcTask Inputs/GVL_Sensor.stGraniteR.iRawCnts <-> AI Standard Channel 1/Value
//   Motion/Motion Instance <-> CX2020 (EtherCAT)/Term 1 (EK1200)/Term 2 (EK1122)/Rack#2B-01 Coupler (EK1100)/Rack#2B-04 PS_P (EL3064)
//     PlcTask Inputs/GVL_Sensor.stPS1.iRawCnts <-> AI Standard Channel 1/Value
//     PlcTask Inputs/GVL_Sensor.stPS2.iRawCnts <-> AI Standard Channel 2/Value
//     PlcTask Inputs/GVL_Sensor.stPS3.iRawCnts <-> AI Standard Channel 3/Value
//   Motion/Motion Instance <-> CX2020 (EtherCAT)/Term 1 (EK1200)/Term 2 (EK1122)/Rack#2B-01 Coupler (EK1100)/Rack#2B-05 SV_AIR (EL2004)
//     PlcTask Outputs/GVL_Main.bOpenSV1 <-> Channel 1/Output
//     PlcTask Outputs/GVL_Main.bOpenSV2 <-> Channel 2/Output
//   Motion/Motion Instance <-> CX2020 (EtherCAT)/Term 1 (EK1200)/Term 2 (EK1122)/Rack#2B-01 Coupler (EK1100)/Rack#2B-07 ENC_X1_X2 (EL5042)
//     PlcTask Inputs/GVL_Main.M3.nRawEncoderULINT <-> FB Inputs Channel 1/Position
//     PlcTask Inputs/GVL_Main.M4.nRawEncoderULINT <-> FB Inputs Channel 2/Position
//   Motion/Motion Instance <-> CX2020 (EtherCAT)/Term 1 (EK1200)/Term 2 (EK1122)/Rack#2B-01 Coupler (EK1100)/Rack#2B-08 ENC_Y1_Y2 (EL5042)
//     PlcTask Inputs/GVL_Main.M5.nRawEncoderULINT <-> FB Inputs Channel 1/Position
//     PlcTask Inputs/GVL_Main.M6.nRawEncoderULINT <-> FB Inputs Channel 1/Position
